       "InstE2MenergyMeterDriver".driverData.pL1Min := 0.0;
       "InstE2MenergyMeterDriver".driverData.pL1Max := 0.0;
       "InstE2MenergyMeterDriver".driverData.pL2Min := 0.0;
       "InstE2MenergyMeterDriver".driverData.pL2Max := 0.0;
       "InstE2MenergyMeterDriver".driverData.pL3Min := 0.0;
       "InstE2MenergyMeterDriver".driverData.pL3Max := 0.0;

       "InstE2MenergyMeterDriver".driverData.qL1Min := 0.0;
       "InstE2MenergyMeterDriver".driverData.qL1Max := 0.0;
       "InstE2MenergyMeterDriver".driverData.qL2Min := 0.0;
       "InstE2MenergyMeterDriver".driverData.qL2Max := 0.0;
       "InstE2MenergyMeterDriver".driverData.qL3Min := 0.0;
       "InstE2MenergyMeterDriver".driverData.qL3Max := 0.0;

   END_IF;

   "Unit1.EmNodes".powerMeter := "InstE2MenergyMeterDriver".driverData;
END_REGION

REGION Network 4: Routing AI_EnergyMeter data to HMI interface
   // Call of Lsicar_EnMeterDataToHmi FB
   RUNG wire#powerrail
      "InstEmDataHmi"(energyMeter01Visu := "InstE2MenergyMeterDriver".driverData, energyMeter02Visu :=, energyMeter03Visu :=, energyMeter04Visu :=, energyMeter05Visu :=, energyMeter06Visu :=, energyMeter07Visu :=, energyMeter08Visu :=)
   END_RUNG
   // the same network as SCL:
   "InstEmDataHmi"(energyMeter01Visu := "InstE2MenergyMeterDriver".driverData);   // "LSicar_EnMeterDataToHmi"
END_REGION
END_FUNCTION

FUNCTION "CallEnEffMonitor" : Void   // FC32, LAD
TITLE = CallEnergyEfficencyMonitor
AUTHOR : SICAR
FAMILY : Energy_EEM
VERSION : 1.0
// The S7 Energy Efficiency-Monitor (or S7 EE-Monitor) allows you to record the energy consumption of your machine in a SIMATIC controller, and to analyze the results on the basis of the energy and media requirements.
// stored: IsIECCheckEnabled true, SetENOAutomatically true
   VAR_TEMP
      tempMeasPointIndex : USInt;   // HMI index
      tempCycleCounterAvgCalc : DInt;   // Calculation to TOD
      tempPlantInProduction : Bool;   // Plant in production
      tempReturnValue : Int;   // Temporärer Wert zur Speicherung der EnPi-Resetzeit
   END_VAR
   // Ret_Val : Ret_Val
   VAR_TEMP   // added for the SCL form of the ladder/FBD networks
      _w1 : Bool;
      _w2 : Bool;
      _w3 : Bool;
      _w4 : Bool;
   END_VAR
BEGIN

REGION Network 1: BLOCK INFO HEADER
   // SIEMENS AG / (c)Copyright 2023
   // ------------------------------------------------------------------------------
   // Title:            CallEnEffMonitor (FC32)
   // Comment/Function: Call of Demo EnergyMeter and Energy Efficient M for EEMM demonstration
   // Library/Family:   Energy
   // Author:           SICAR
   // Tested with:      ---
   // Engineering:      TIA Portal V19
   // Restrictions:     -
   // Requirements:     ---
   // ------------------------------------------------------------------------------
   // Change log table:
   // Version  | Date       | Expert in charge       | Changes applied
   // ---------|------------|------------------------|------------------------------
   // 05.00.00 | 01.09.2023 | SICAR
   //                         First released version
END_REGION

REGION Network 2: DESCRIPTION
   // The Energy Efficiency Monitor “EEM” integrated in SICAR is based on the application example in entry ID: 109753230 V1.0 dated 02/2018 of the Siemens Industry Online Support, see: 
   // 
   // https://support.industry.siemens.com/cs/document/109753230/-s7-energy-efficiency-monitor-for-machines?dti=0&lc=en-WW 
   // 
   // **License**  
   // The software package has to be licensed. The necessary license key has to be entered in the data block for energy data “EEmData”, in the array item “licenseKey”. 
   //  
   // {.pageWidth}
   // ![Image](EemEnPiCalc/en/image1.PNG)
   // 
   // The S7 Energy Efficiency-Monitor (or S7 EE-Monitor) allows you to record the energy consumption of your machine in a SIMATIC controller, and to analyze the results on the basis of the energy and media requirements.  
   // https://support.industry.siemens.com/cs/document/109753230/s7-energieeffizienz-monitor-für-maschinen?dti=0&lc=de-WW 
   // 
   // **PLC Data types**  
   //  LSicar_typeEeMenPiCalc 
   //  LSicar_typeEeMenPiEstate 
   //  LSicar_typeEeMenPiLimit 
   //  typeEnMeterOutputData 
   //  typeMeasDataProfileE3 
   //  
   // **WinCC Faceplates**  
   // 
   // ![Image](EemEnPiCalc/en/image3.PNG)
   // 
   // **WinCC Screen**  
   //  
   // ![Image](EemEnPiCalc/en/image4.PNG)
   //  
   // # Devices & networks 
   // 
   // An additional AI Energy Meter has been added and configured in the SICAR project. The user data has been  
   // configured as module version “EE@Industry measured data profile e3”.  
   // 
   // Select the module version according to your requirements. The data assignment in the FC blocks has to be adjusted according to the selected module version. 
   // 
   // ![Image](EemEnPiCalc/en/image5.PNG)
   //  
   //  
   // 
   //  #### PLC Programm blocks 
   // 
   // ##### CallEnSeem  
   // The block is called in OB “CYCLIC_INTERRUPT_100MS_OB” (100ms cycle). The block contains the following instructions which can be found in “Instructions > Optional packages > Energy Suite extensions”.
   // 
   // **EnS_EEm_Calc:**  
   // The instruction calculates operating state-related energy data of machines and plants for uniform efficiency evaluation, in accordance with the VDMA 34179 measuring directive. 
   // 
   // ---
   // Note
   // :     The instruction calculates the energy efficiency value of the respective state for up to 8 operating states, and the global energy efficiency value. 
   // :     The maximum number of configurable measuring points is 10. Refer to the documentation of the entry ID. 
   // 
   // ---
   // 
   // **EnS_EEm_Report:**  
   // The instruction writes the data for the efficiency report to the data log on the SIMATIC memory card, in accordance with the VDMA 34179 measuring directive. The data log is a CSV file. 
   // 
   // ##### CallEnEffMonitor
   // ---
   // Note
   // :     The assignment of the readings as well as the formation of additional signals can be represented only exemplarily here. It has to be adapted to the actual plant conditions! 
   // 
   // ---
   // 
   // * Networks 1 & 2: The readings of the two AI-Energy-Meters are entered in the DB “EeMonitor”, in an array [0..9] in accordance with the measurement data profile “typeMeasDataProfileE3”. 
   // * Network 3: According to the selection of a measuring point on the HMI, data of the respective measuring point is routed to the HMI data area. The selection is done with a Pull-Down menu and a symbolic I/O field. 
   // * Network 4: Several tags in the EnS…data types are not marked as accessible / visible. In order to display these tags on the HMI all the same, they are routed to DB “EeMonitor” in structure “typeEnMeterWorkHmi”. There the tags are marked as accessible / visible.  
   // * Network 5: A collective signal is generated, according to the exemplary calls for OP area 1. This is only an example! The collective signal shows that the plant is producing parts, by a disjunction (OR) of all outputs. If an output is controlled, the plant is moving and producing parts. This collective signal is used later on to generate the energetic states “eState”. A delay of 3 seconds has been configured so that a short break in controlling the outputs will not change the energetic state. *
   // * Network 6: The signals for the energetic states are generated here. 
   // * Network 7: Simulation On/Off: A part counter is simulated here. Note: the simulation can be switched on and off with a button in the screen. 
   // * Network 8: Simulation On/Off. Energy counters for both AI-Energy-Meters are simulated here. Note: the simulation can be switched on and off with a button in the screen. 
   // * Network 9: Call of blocks “EemDemoSimulation” and “EemDemoResetValEMeter”. 
   // * Network 10: Call of block “EemEnPiCalc” and data routing according to the selection of a measuring point on the HMI. 
   // * Network 11: Error evaluation of block “EemEnPiCalc” to generate ProDiag messages. 
   // * Network 12: Error evaluation of block “EnS_EEm_Report” to generate ProDiag messages.  
   // 
   // ##### EemDemoResetValEMeter  
   // 
   // The block resets certain measurement values by controlling the respective outputs in the I/O area of the AI-Energy-Meter. 
   // 
   // ##### EemDemoSimulation  
   // 
   // This block simulates higher or lower energy values, according to the energetic states “eState”. 
   // 
   // ##### EemEnPiCalc
   // This block calculates the ENPI (Energy value Pro Item). It substitutes the script “EEm_EnPI_Efficiency” of the entry ID. 
   // 
   // ---
   // Note
   // :     All block parameters are provided with “pre-defined actual parameters”.
   // 
   // ---
   // 
   // **Operation mode Automatic / Manual**  
   // 
   // The blocks are independent of operation modes. Therefor they are not assigned to any operation mode area. 
   // 
   // **PLC Alarm text list**  
   // 
   // The following PLC alarm text lists have been created: 
   // 
   // * **EEMonitor_Calc_Warn_PD** ProDiag alarm text list for alarms by instruction “EnS_EEm_Calc”.   
   // * **EEMonitor_Report_Warn_PD** ProDiag alarm text list for alarms by instruction “EnS_EEm_Report”.   
   // Both PLC alarm text lists have been entered in the PLC alarm text list “GLOBAL_GENERAL_AlarmTextList”. 
   // 
   // ---
   // Note
   // :     The alarm texts are provided in two languages (German, English). Please consider the multilingual nature of the entries. 
   // 
   // ---
   // 
   // #### PLC Data types 
   // 
   // PLC data types used for PLC program block or HMI faceplate:  
   // ![Image](_Icon/reference.PNG)  See ..\Library Types\LSicar_typeEeMenPiCalc.pdf  
   // 
   // #### WinCC Objects 
   // 
   // **WinCC HMI-tags**  
   // 
   // The HMI tags are stored in the tag table “AI_EnergyMeter_EEM” in the SICAR project.  
   // 
   // **WinCC Text and graphics lists**  
   // 
   // The text list “EE-MONITOR_MEASUREPOINT” contains the texts necessary for the pull-down menu / symbolic I/O field in the screen. Please take into account the multilingual nature of the entries.  
   // 
   // **WinCC Faceplates**  
   // 
   // The faceplates are stored in the project library, in folder “types”. They have been created using several WinCC objects; they are animated depending on the state. 
   // 
   // * EEM_EnPI_EnergyPerItem:	display of ENPI (ENergy Per Item) 
   // * EEM_ViewBar_Diff-AVG-REF:	bar display to compare reference value and average value 
   // * EEM_ViewBar_EState-Total:	bar display of energy status (not used at this time) 
   // * EEM_ViewBarCurve_EState:	Total: bar display and curve display of the energy values  
   // 
   // **WinCC-screen** 
   // 
   // 1. HMI Screens:	EE-MONITOR_ENERGY: display of the energy values 
   // 2. HMI Popup-screens 
   // 	* EEM_LEGEND_Popup: 		Legend 
   // 	* EEM_INFO-MACHINE_Popup: 	Machine information 
   // 	* EEM_STARTMEASURE_Popup: 	Popup to start the normal measurement or the reference measurement  
   // 	* EEM_UIPE_Popup: 		display of voltage, current, power, and energy 
   // 	* MORE_EEM_Popup: 		Popup with additional buttons 
   // 	* MORE_AddOn_Popup: 		supplemented  with button “EE-Monitor” 
   // 
   //  
   // 
   // {.pageWidth}
   // ![Image](EemEnPiCalc/en/image6.PNG)
   //  
   //  
   // 
   // #### Additional information
   // 
   // #### Update info
   // 
   // #### Further documentations
END_REGION

REGION Network 3: select measurement values
   // can be from EnergyMeter driver or directly from any hardware (in this example EnergyMeter module and PAC)
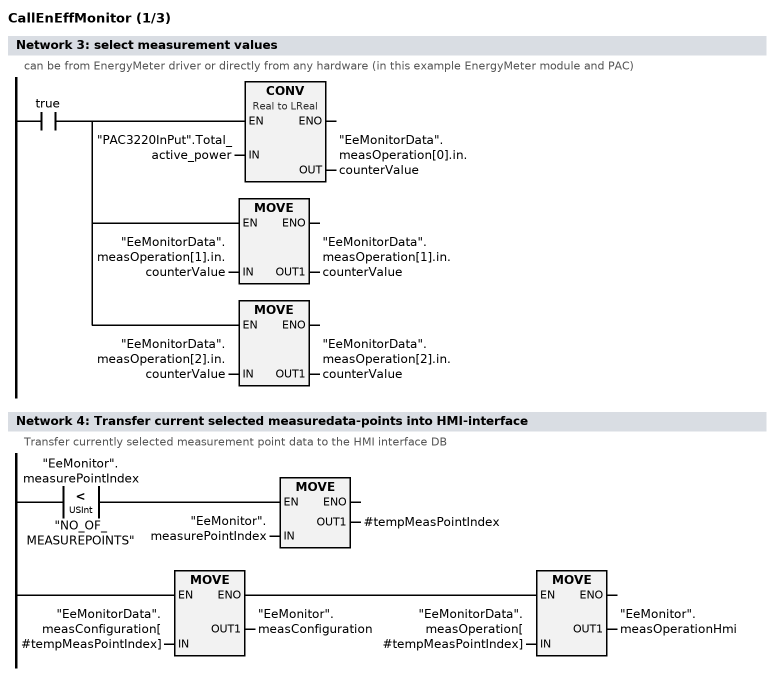
   RUNG wire#powerrail
      Contact( true )
      wire#w1
      { S7_Templates := "[SrcType := Real, DestType := LReal]" } Convert(in := "PAC3220InPut".Total_active_power, out => "EeMonitorData".measOperation[0].in.counterValue)
   END_RUNG
   RUNG wire#w1
      Move(in := "EeMonitorData".measOperation[1].in.counterValue, out1 => "EeMonitorData".measOperation[1].in.counterValue)
   END_RUNG
   RUNG wire#w1
      Move(in := "EeMonitorData".measOperation[2].in.counterValue, out1 => "EeMonitorData".measOperation[2].in.counterValue)
   END_RUNG
   // the same network as SCL:
   IF true THEN
       "EeMonitorData".measOperation[0].in.counterValue := REAL_TO_LREAL("PAC3220InPut".Total_active_power);
       "EeMonitorData".measOperation[1].in.counterValue := "EeMonitorData".measOperation[1].in.counterValue;
       "EeMonitorData".measOperation[2].in.counterValue := "EeMonitorData".measOperation[2].in.counterValue;
   END_IF;
END_REGION

REGION Network 4: Transfer current selected measuredata-points into HMI-interface
   // Transfer currently selected measurement point data to the HMI interface DB
   RUNG wire#powerrail
      { S7_Templates := "SrcType := USInt" } LT_Contact(in1 := "EeMonitor".measurePointIndex, in2 := "NO_OF_MEASUREPOINTS")
      Move(in := "EeMonitor".measurePointIndex, out1 => #tempMeasPointIndex)
   END_RUNG
   RUNG wire#powerrail
      Move(in := "EeMonitorData".measConfiguration[#tempMeasPointIndex], out1 => "EeMonitor".measConfiguration)
      Move(in := "EeMonitorData".measOperation[#tempMeasPointIndex], out1 => "EeMonitor".measOperationHmi)
   END_RUNG
   // the same network as SCL:
   IF "EeMonitor".measurePointIndex < "NO_OF_MEASUREPOINTS" THEN
       #tempMeasPointIndex := "EeMonitor".measurePointIndex;
   END_IF;
   "EeMonitor".measConfiguration := "EeMonitorData".measConfiguration[#tempMeasPointIndex];
   "EeMonitor".measOperationHmi := "EeMonitorData".measOperation[#tempMeasPointIndex];
END_REGION

REGION Network 5: WORKaround: Transfer data from EeMonitroData to EeMonitor.work
   // Convertion of Time to DTL and adding time zone with date and time taken from EnS_EEm_Calc for representing the actual date and time in the current country.
   // Data is copied from EeMonitorData to EeMonitor.work
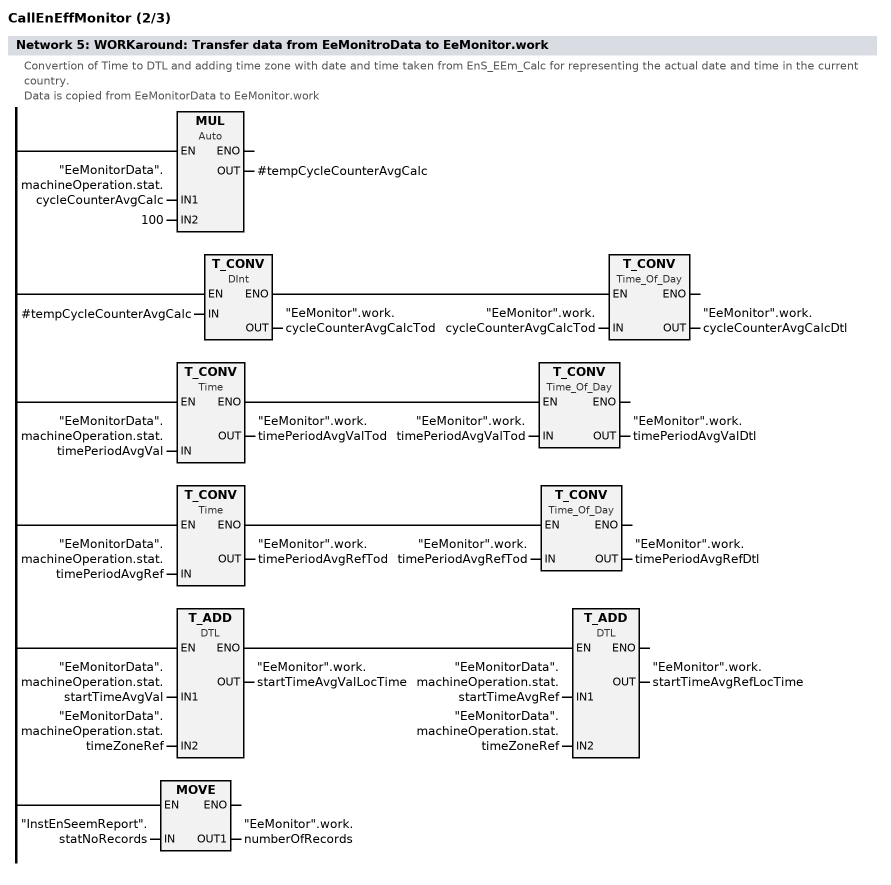
   RUNG wire#powerrail
      Mul(in1 := "EeMonitorData".machineOperation.stat.cycleCounterAvgCalc, in2 := 100, out => #tempCycleCounterAvgCalc)
   END_RUNG
   RUNG wire#powerrail
      { S7_Templates := "[src_type := DInt, dest_type := Time_Of_Day]" } T_CONV(IN := #tempCycleCounterAvgCalc, OUT => "EeMonitor".work.cycleCounterAvgCalcTod)
      { S7_Templates := "[src_type := Time_Of_Day, dest_type := DTL]" } T_CONV(IN := "EeMonitor".work.cycleCounterAvgCalcTod, OUT => "EeMonitor".work.cycleCounterAvgCalcDtl)
   END_RUNG
   RUNG wire#powerrail
      { S7_Templates := "[src_type := Time, dest_type := Time_Of_Day]" } T_CONV(IN := "EeMonitorData".machineOperation.stat.timePeriodAvgVal, OUT => "EeMonitor".work.timePeriodAvgValTod)
      { S7_Templates := "[src_type := Time_Of_Day, dest_type := DTL]" } T_CONV(IN := "EeMonitor".work.timePeriodAvgValTod, OUT => "EeMonitor".work.timePeriodAvgValDtl)
   END_RUNG
   RUNG wire#powerrail
      { S7_Templates := "[src_type := Time, dest_type := Time_Of_Day]" } T_CONV(IN := "EeMonitorData".machineOperation.stat.timePeriodAvgRef, OUT => "EeMonitor".work.timePeriodAvgRefTod)
      { S7_Templates := "[src_type := Time_Of_Day, dest_type := DTL]" } T_CONV(IN := "EeMonitor".work.timePeriodAvgRefTod, OUT => "EeMonitor".work.timePeriodAvgRefDtl)
   END_RUNG
   RUNG wire#powerrail
      { S7_Templates := "[date_type := DTL, time_type := Time]" } T_ADD(IN1 := "EeMonitorData".machineOperation.stat.startTimeAvgVal, IN2 := "EeMonitorData".machineOperation.stat.timeZoneRef, OUT => "EeMonitor".work.startTimeAvgValLocTime)
      { S7_Templates := "[date_type := DTL, time_type := Time]" } T_ADD(IN1 := "EeMonitorData".machineOperation.stat.startTimeAvgRef, IN2 := "EeMonitorData".machineOperation.stat.timeZoneRef, OUT => "EeMonitor".work.startTimeAvgRefLocTime)
   END_RUNG
   RUNG wire#powerrail
      Move(in := "InstEnSeemReport".statNoRecords, out1 => "EeMonitor".work.numberOfRecords)
   END_RUNG
   // the same network as SCL:
   #tempCycleCounterAvgCalc := "EeMonitorData".machineOperation.stat.cycleCounterAvgCalc * 100;
   T_CONV(IN := #tempCycleCounterAvgCalc, OUT => "EeMonitor".work.cycleCounterAvgCalcTod, ENO => #_w1);
   IF #_w1 THEN
       T_CONV(IN := "EeMonitor".work.cycleCounterAvgCalcTod, OUT => "EeMonitor".work.cycleCounterAvgCalcDtl);
   END_IF;
   T_CONV(IN := "EeMonitorData".machineOperation.stat.timePeriodAvgVal,
          OUT => "EeMonitor".work.timePeriodAvgValTod,
          ENO => #_w2);
   IF #_w2 THEN
       T_CONV(IN := "EeMonitor".work.timePeriodAvgValTod, OUT => "EeMonitor".work.timePeriodAvgValDtl);
   END_IF;
   T_CONV(IN := "EeMonitorData".machineOperation.stat.timePeriodAvgRef,
          OUT => "EeMonitor".work.timePeriodAvgRefTod,
          ENO => #_w3);
   IF #_w3 THEN
       T_CONV(IN := "EeMonitor".work.timePeriodAvgRefTod, OUT => "EeMonitor".work.timePeriodAvgRefDtl);
   END_IF;
   T_ADD(IN1 := "EeMonitorData".machineOperation.stat.startTimeAvgVal,
         IN2 := "EeMonitorData".machineOperation.stat.timeZoneRef,
         OUT => "EeMonitor".work.startTimeAvgValLocTime,
         ENO => #_w4);
   IF #_w4 THEN
       T_ADD(IN1 := "EeMonitorData".machineOperation.stat.startTimeAvgRef,
             IN2 := "EeMonitorData".machineOperation.stat.timeZoneRef,
             OUT => "EeMonitor".work.startTimeAvgRefLocTime);
   END_IF;
   "EeMonitor".work.numberOfRecords := "InstEnSeemReport".statNoRecords;
END_REGION

REGION Network 6: Operation modes to "eState"
   // Sets Estate number accoriding to the selected state
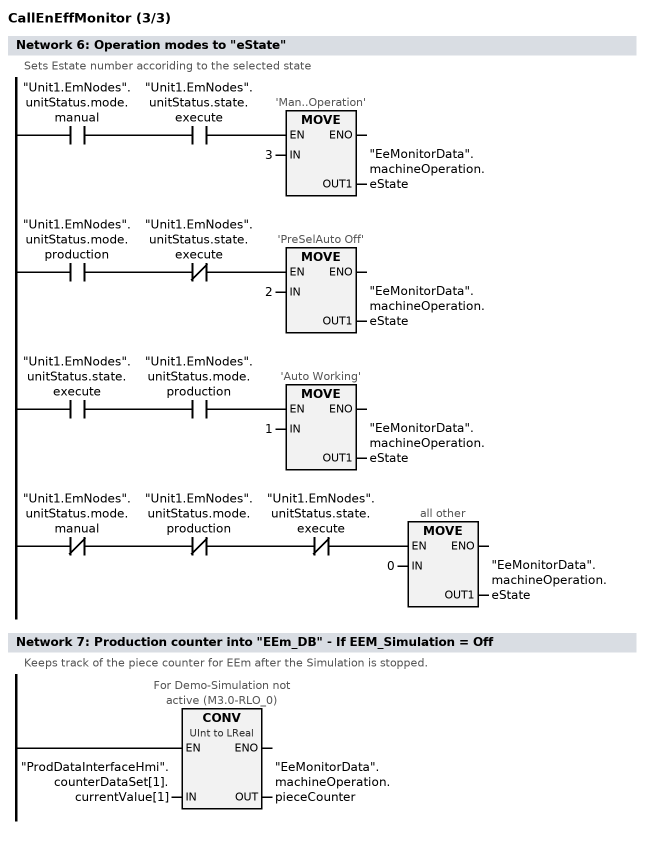
   RUNG wire#powerrail
      Contact( "Unit1.EmNodes".unitStatus.mode.manual )
      Contact( "Unit1.EmNodes".unitStatus.state.execute )
      Move(in := 3, out1 => "EeMonitorData".machineOperation.eState)   // 'Man..Operation'
   END_RUNG
   RUNG wire#powerrail
      Contact( "Unit1.EmNodes".unitStatus.mode.production )
      I_Contact( "Unit1.EmNodes".unitStatus.state.execute )
      Move(in := 2, out1 => "EeMonitorData".machineOperation.eState)   // 'PreSelAuto Off'
   END_RUNG
   RUNG wire#powerrail
      Contact( "Unit1.EmNodes".unitStatus.state.execute )
      Contact( "Unit1.EmNodes".unitStatus.mode.production )
      Move(in := 1, out1 => "EeMonitorData".machineOperation.eState)   // 'Auto Working'
   END_RUNG
   RUNG wire#powerrail
      I_Contact( "Unit1.EmNodes".unitStatus.mode.manual )
      I_Contact( "Unit1.EmNodes".unitStatus.mode.production )
      I_Contact( "Unit1.EmNodes".unitStatus.state.execute )
      Move(in := 0, out1 => "EeMonitorData".machineOperation.eState)   // all other
   END_RUNG
   // the same network as SCL:
   IF "Unit1.EmNodes".unitStatus.mode.manual AND "Unit1.EmNodes".unitStatus.state.execute THEN
       "EeMonitorData".machineOperation.eState := 3;   // 'Man..Operation'
   END_IF;
   IF "Unit1.EmNodes".unitStatus.mode.production AND NOT "Unit1.EmNodes".unitStatus.state.execute THEN
       "EeMonitorData".machineOperation.eState := 2;   // 'PreSelAuto Off'
   END_IF;
   IF "Unit1.EmNodes".unitStatus.state.execute AND "Unit1.EmNodes".unitStatus.mode.production THEN
       "EeMonitorData".machineOperation.eState := 1;   // 'Auto Working'
   END_IF;
   IF NOT "Unit1.EmNodes".unitStatus.mode.manual AND NOT "Unit1.EmNodes".unitStatus.mode.production AND NOT "Unit1.EmNodes".unitStatus.state.execute THEN
       "EeMonitorData".machineOperation.eState := 0;   // all other
   END_IF;
END_REGION

REGION Network 7: Production counter into "EEm_DB" - If EEM_Simulation = Off
   // Keeps track of the piece counter for EEm after the Simulation is stopped.
   RUNG wire#powerrail
      { S7_Templates := "[SrcType := UInt, DestType := LReal]" } Convert(in := "ProdDataInterfaceHmi".counterDataSet[1].currentValue[1], out => "EeMonitorData".machineOperation.pieceCounter)   // For Demo-Simulation not active (M3.0-RLO_0)
   END_RUNG
   // the same network as SCL:
   "EeMonitorData".machineOperation.pieceCounter := UINT_TO_LREAL("ProdDataInterfaceHmi".counterDataSet[1].currentValue[1]);   // For Demo-Simulation not active (M3.0-RLO_0)
END_REGION

REGION Network 8 (SCL): Reset EnPI values
   // Reads the current time and store it to provide the user the information about the last EnPi reset
   // Check for the trigger to reset/recalculate the EnPI values
   IF ("EeMonitorData".internalData.enpiResetTrigger = TRUE) THEN

       // Read the current time and store it to provide the user the information
       // about the last reset
       #tempReturnValue := RD_LOC_T("EeMonitorData".internalData.enpiResetTime);

       // Reset the trigger
       "EeMonitorData".internalData.enpiResetTrigger := FALSE;
   ELSE
       ; // No trigger
   END_IF;
END_REGION
END_FUNCTION

FUNCTION "CallSettings" : Void   // FC8, LAD
// Call of settings blocks
// stored: IsIECCheckEnabled true, SetENOAutomatically false
BEGIN

REGION Network 1: BLOCK INFO HEADER
   // SIEMENS AG / (c)Copyright 2023
   // ------------------------------------------------------------------------------
   // Title:            CallSettings
   // Comment/Function: Call of SICAR Settings blocks
   // Library/Family:   -
   // Author:           -
   // Tested with:      ---
   // Engineering:      TIA Portal V19
   // Restrictions:     -
   // Requirements:     ---
   // ------------------------------------------------------------------------------
   // Change log table:
   // Version | Date | Expert in charge | Changes applied
   // -------|---------|-------------|--------------------------------------------
   // 01.00.00 | 01.01.1999 | Person x | First released version
   // 01.00.01 | 02.01.1999 | Person y | Block was Updated
END_REGION

REGION Network 2: Set set PLC date and time
   // Change local date and time of the PLC
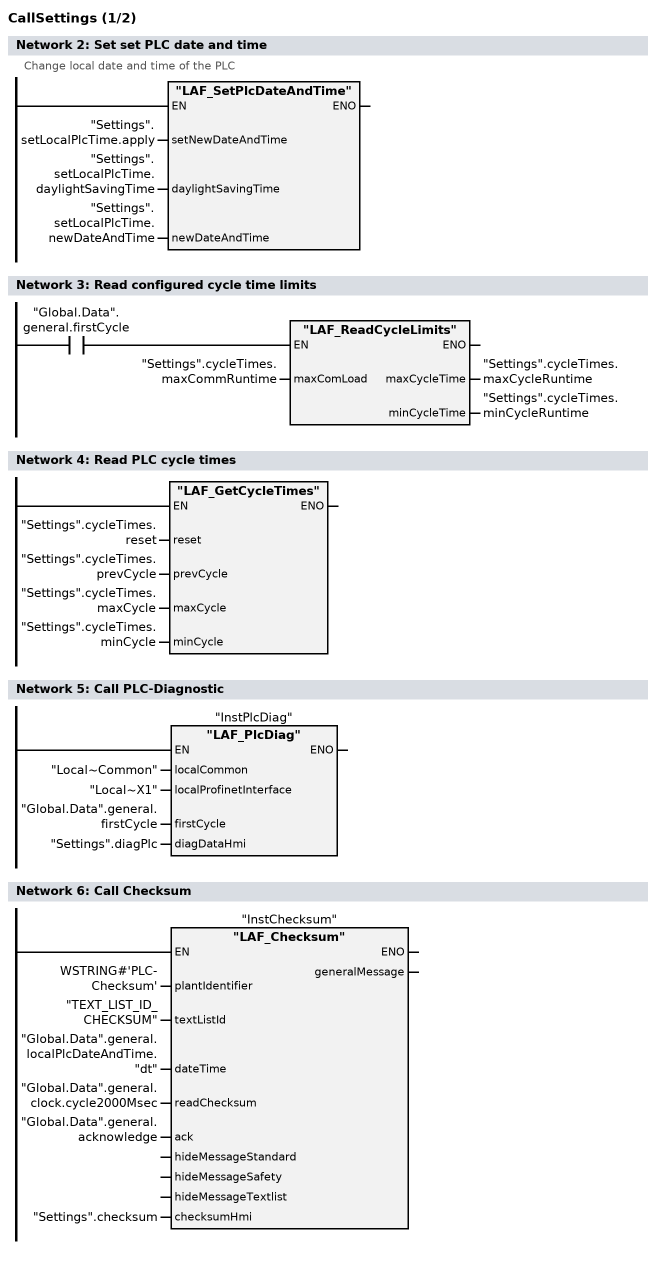
   RUNG wire#powerrail
      "LAF_SetPlcDateAndTime"(setNewDateAndTime := "Settings".setLocalPlcTime.apply, daylightSavingTime := "Settings".setLocalPlcTime.daylightSavingTime, newDateAndTime := "Settings".setLocalPlcTime.newDateAndTime)
   END_RUNG
   // the same network as SCL:
   "LAF_SetPlcDateAndTime"(setNewDateAndTime := "Settings".setLocalPlcTime.apply,
                           daylightSavingTime := "Settings".setLocalPlcTime.daylightSavingTime,
                           newDateAndTime := "Settings".setLocalPlcTime.newDateAndTime);
END_REGION

REGION Network 3: Read configured cycle time limits
   RUNG wire#powerrail
      Contact( "Global.Data".general.firstCycle )
      "LAF_ReadCycleLimits"(maxComLoad := "Settings".cycleTimes.maxCommRuntime, maxCycleTime => "Settings".cycleTimes.maxCycleRuntime, minCycleTime => "Settings".cycleTimes.minCycleRuntime)
   END_RUNG
   // the same network as SCL:
   IF "Global.Data".general.firstCycle THEN
       "LAF_ReadCycleLimits"(maxComLoad := "Settings".cycleTimes.maxCommRuntime,
                             maxCycleTime => "Settings".cycleTimes.maxCycleRuntime,
                             minCycleTime => "Settings".cycleTimes.minCycleRuntime);
   END_IF;
END_REGION

REGION Network 4: Read PLC cycle times
   RUNG wire#powerrail
      "LAF_GetCycleTimes"(reset := "Settings".cycleTimes.reset, prevCycle := "Settings".cycleTimes.prevCycle, maxCycle := "Settings".cycleTimes.maxCycle, minCycle := "Settings".cycleTimes.minCycle)
   END_RUNG
   // the same network as SCL:
   "LAF_GetCycleTimes"(reset := "Settings".cycleTimes.reset,
                       prevCycle := "Settings".cycleTimes.prevCycle,
                       maxCycle := "Settings".cycleTimes.maxCycle,
                       minCycle := "Settings".cycleTimes.minCycle);
END_REGION

REGION Network 5: Call PLC-Diagnostic
   RUNG wire#powerrail
      "InstPlcDiag"(localCommon := "Local~Common", localProfinetInterface := "Local~X1", firstCycle := "Global.Data".general.firstCycle, diagDataHmi := "Settings".diagPlc)
   END_RUNG
   // the same network as SCL:
   "InstPlcDiag"(localCommon := "Local~Common",   // "LAF_PlcDiag"
                 localProfinetInterface := "Local~X1",
                 firstCycle := "Global.Data".general.firstCycle,
                 diagDataHmi := "Settings".diagPlc);
END_REGION

REGION Network 6: Call Checksum
   RUNG wire#powerrail
      "InstChecksum"(plantIdentifier := WSTRING#'PLC-Checksum', textListId := "TEXT_LIST_ID_CHECKSUM", dateTime := "Global.Data".general.localPlcDateAndTime."dt", readChecksum := "Global.Data".general.clock.cycle2000Msec, ack := "Global.Data".general.acknowledge, hideMessageStandard :=, hideMessageSafety :=, hideMessageTextlist :=, checksumHmi := "Settings".checksum, generalMessage =>)
   END_RUNG
   // the same network as SCL:
   "InstChecksum"(plantIdentifier := WSTRING#'PLC-Checksum',   // "LAF_Checksum"
                  textListId := "TEXT_LIST_ID_CHECKSUM",
                  dateTime := "Global.Data".general.localPlcDateAndTime."dt",
                  readChecksum := "Global.Data".general.clock.cycle2000Msec,
                  ack := "Global.Data".general.acknowledge,
                  checksumHmi := "Settings".checksum);
END_REGION

REGION Network 7: Call SMC-Diagnostic (SIMATIC Memory Card - Diagnostic)
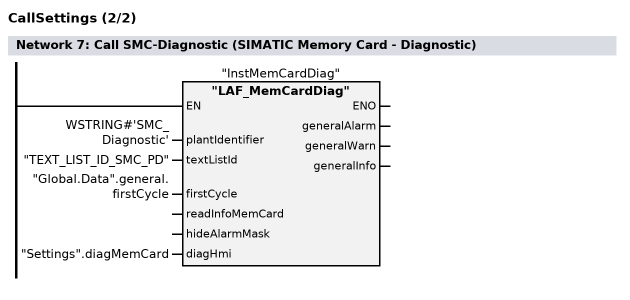
   RUNG wire#powerrail
      "InstMemCardDiag"(plantIdentifier := WSTRING#'SMC_Diagnostic', textListId := "TEXT_LIST_ID_SMC_PD", firstCycle := "Global.Data".general.firstCycle, readInfoMemCard :=, hideAlarmMask :=, diagHmi := "Settings".diagMemCard, generalAlarm =>, generalWarn =>, generalInfo =>)
   END_RUNG
   // the same network as SCL:
   "InstMemCardDiag"(plantIdentifier := WSTRING#'SMC_Diagnostic',   // "LAF_MemCardDiag"
                     textListId := "TEXT_LIST_ID_SMC_PD",
                     firstCycle := "Global.Data".general.firstCycle,
                     diagHmi := "Settings".diagMemCard);
END_REGION
END_FUNCTION

ORGANIZATION_BLOCK "DiagnosticErrorInterrupt"   // OB82, LAD, DiagnosticErrorInterrupt
// stored: SetENOAutomatically false
   VAR_INPUT
      IO_State : Word;   // IO state of the HW object
      LADDR : HW_ANY;   // Hardware identifier
      Channel : UInt;   // Channel number
      MultiError : Bool;   // =true if more than one error is present
   END_VAR
BEGIN
END_ORGANIZATION_BLOCK

ORGANIZATION_BLOCK "HardwareInterrupt"   // OB40, LAD, HardwareInterrupt
// stored: SetENOAutomatically false
   VAR_INPUT
      LADDR : HW_IO;   // Hardware identifier
      USI : Word;   // User structure identifier
      IChannel : USInt;   // Interrupt channel number
      EventType : Byte;   // EventType
      PointAddr : DWord;
   END_VAR
BEGIN
END_ORGANIZATION_BLOCK

ORGANIZATION_BLOCK "IO_AccessError"   // OB122, LAD, IOAccessError
// stored: SetENOAutomatically false
   VAR_INPUT
      BlockNr : UInt;   // Number of causing block
      Reaction : USInt;   // 0:ignore, 1:substitute, 2:skip
      Fault_ID : Byte;   // 16#42:reading, 16#43:writing
      BlockType : USInt;   // 16#01:OB, 16#02:FC, 16#03:FB, 16#04:SFC, 16#05:SFB, 16#06:DB: Type of block causing the error
      Area : USInt;   // 16#81:I, 16#82:Q: IO area where the IOaccess error occured
      DBNr : DB_ANY;   // Reserved for system
      Csg_OBNr : OB_ANY;   // Number of OB causing the error
      Csg_Prio : USInt;   // Priority of OB causing the error
      Width : USInt;   // 0:bit, 1:byte, 2:word, 3:dword, 4:lword
   END_VAR
BEGIN
END_ORGANIZATION_BLOCK

ORGANIZATION_BLOCK "Interrupt1s"   // OB31, LAD, CyclicInterrupt
TITLE = Cyclic interrupt 100ms
AUTHOR : SICAR
FAMILY : OB
VERSION : 1.0
// organisation block
// stored: IsIECCheckEnabled true, SetENOAutomatically true
   VAR_INPUT
      Initial_Call : Bool;   // Initial call of this OB
      Event_Count : Int;   // Events discarded
   END_VAR
BEGIN

REGION Network 1: ChangeLog
   // Change log table:
   // Version | Date | Expert in charge | Changes applied
   // -------|---------|-------------|--------------------------------------------
   // 01.00.00 | 01.01.1999 | Person x | First released version
   // 01.00.01 | 02.01.1999 | Person y | Block was Updated
END_REGION

REGION Network 2: Call & measure-data into "EEmData_DB"
   // Call the energy efficiency monitor functions
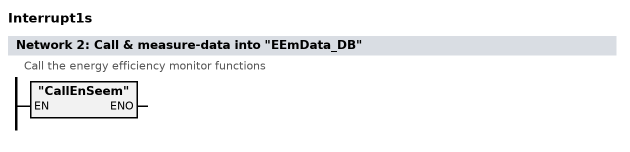
   RUNG wire#powerrail
      "CallEnSeem"()
   END_RUNG
   // the same network as SCL:
   "CallEnSeem"();
END_REGION
END_ORGANIZATION_BLOCK

FUNCTION "CallEnSeem" : Void   // FC34, LAD
TITLE = CallEnSeem
AUTHOR : SICAR
FAMILY : Energy_EEM
VERSION : 1.0
// The S7 Energy Efficiency-Monitor (or S7 EE-Monitor) allows you to record the energy consumption of your machine in a SIMATIC controller, and to analyze the results on the basis of the energy and media requirements.
// stored: IsIECCheckEnabled true, SetENOAutomatically true
   // Ret_Val : Ret_Val
BEGIN

REGION Network 1: BLOCK INFO HEADER
   // SIEMENS AG / (c)Copyright 2023
   // ------------------------------------------------------------------------------
   // Title:            CallEnSeem (FC34)
   // Comment/Function: The S7 Energy Efficiency-Monitor (or S7 EE-Monitor) allows you to record the energy consumption of your machine in a SIMATIC controller, and to analyze the results on the basis of the energy and media requirements.
   // Library/Family:   Energy_EEM
   // Author:           SICAR
   // Tested with:      ---
   // Engineering:      TIA Portal V19
   // Restrictions:     -
   // Requirements:     ---
   // ------------------------------------------------------------------------------
   // Change log table:
   // Version | Date | Expert in charge | Changes applied
   // -------|---------|-------------|--------------------------------------------
   // 01.00.00 | 01.01.1999 | Person x | First released version
   // 01.00.01 | 02.01.1999 | Person y | Block was Updated
END_REGION

REGION Network 2: DESCRIPTION
   // The Energy Efficiency Monitor “EEM” integrated in SICAR is based on the application example in entry ID: 109753230 V1.0 dated 02/2018 of the Siemens Industry Online Support, see: 
   // 
   // https://support.industry.siemens.com/cs/document/109753230/-s7-energy-efficiency-monitor-for-machines?dti=0&lc=en-WW 
   // 
   // **License**  
   // The software package has to be licensed. The necessary license key has to be entered in the data block for energy data “EEmData”, in the array item “licenseKey”. 
   //  
   // {.pageWidth}
   // ![Image](EemEnPiCalc/en/image1.PNG)
   // 
   // The S7 Energy Efficiency-Monitor (or S7 EE-Monitor) allows you to record the energy consumption of your machine in a SIMATIC controller, and to analyze the results on the basis of the energy and media requirements.  
   // https://support.industry.siemens.com/cs/document/109753230/s7-energieeffizienz-monitor-für-maschinen?dti=0&lc=de-WW 
   // 
   // **PLC Data types**  
   //  LSicar_typeEeMenPiCalc 
   //  LSicar_typeEeMenPiEstate 
   //  LSicar_typeEeMenPiLimit 
   //  typeEnMeterOutputData 
   //  typeMeasDataProfileE3 
   //  
   // **WinCC Faceplates**  
   // 
   // ![Image](EemEnPiCalc/en/image3.PNG)
   // 
   // **WinCC Screen**  
   //  
   // ![Image](EemEnPiCalc/en/image4.PNG)
   //  
   // # Devices & networks 
   // 
   // An additional AI Energy Meter has been added and configured in the SICAR project. The user data has been  
   // configured as module version “EE@Industry measured data profile e3”.  
   // 
   // Select the module version according to your requirements. The data assignment in the FC blocks has to be adjusted according to the selected module version. 
   // 
   // ![Image](EemEnPiCalc/en/image5.PNG)
   //  
   //  
   // 
   // #### PLC Programm blocks 
   // 
   // ##### CallEnSeem  
   // The block is called in OB “CYCLIC_INTERRUPT_100MS_OB” (100ms cycle). The block contains the following instructions which can be found in “Instructions > Optional packages > Energy Suite extensions”.
   // 
   // **EnS_EEm_Calc:**  
   // The instruction calculates operating state-related energy data of machines and plants for uniform efficiency evaluation, in accordance with the VDMA 34179 measuring directive. 
   // 
   // ---
   // Note
   // :     The instruction calculates the energy efficiency value of the respective state for up to 8 operating states, and the global energy efficiency value. 
   // :     The maximum number of configurable measuring points is 10. Refer to the documentation of the entry ID. 
   // 
   // ---
   // 
   // **EnS_EEm_Report:**  
   // The instruction writes the data for the efficiency report to the data log on the SIMATIC memory card, in accordance with the VDMA 34179 measuring directive. The data log is a CSV file. 
   // 
   // #### CallEnEffMonitor
   // ---
   // Note
   // :     The assignment of the readings as well as the formation of additional signals can be represented only exemplarily here. It has to be adapted to the actual plant conditions! 
   // 
   // ---
   // 
   // * Networks 1 & 2: The readings of the two AI-Energy-Meters are entered in the DB “EeMonitor”, in an array [0..9] in accordance with the measurement data profile “typeMeasDataProfileE3”. 
   // * Network 3: According to the selection of a measuring point on the HMI, data of the respective measuring point is routed to the HMI data area. The selection is done with a Pull-Down menu and a symbolic I/O field. 
   // * Network 4: Several tags in the EnS…data types are not marked as accessible / visible. In order to display these tags on the HMI all the same, they are routed to DB “EeMonitor” in structure “typeEnMeterWorkHmi”. There the tags are marked as accessible / visible.  
   // * Network 5: A collective signal is generated, according to the exemplary calls for OP area 1. This is only an example! The collective signal shows that the plant is producing parts, by a disjunction (OR) of all outputs. If an output is controlled, the plant is moving and producing parts. This collective signal is used later on to generate the energetic states “eState”. A delay of 3 seconds has been configured so that a short break in controlling the outputs will not change the energetic state. *
   // * Network 6: The signals for the energetic states are generated here. 
   // * Network 7: Simulation On/Off: A part counter is simulated here. Note: the simulation can be switched on and off with a button in the screen. 
   // * Network 8: Simulation On/Off. Energy counters for both AI-Energy-Meters are simulated here. Note: the simulation can be switched on and off with a button in the screen. 
   // * Network 9: Call of blocks “EemDemoSimulation” and “EemDemoResetValEMeter”. 
   // * Network 10: Call of block “EemEnPiCalc” and data routing according to the selection of a measuring point on the HMI. 
   // * Network 11: Error evaluation of block “EemEnPiCalc” to generate ProDiag messages. 
   // * Network 12: Error evaluation of block “EnS_EEm_Report” to generate ProDiag messages.  
   // 
   // #### EemDemoResetValEMeter  
   // 
   // The block resets certain measurement values by controlling the respective outputs in the I/O area of the AI-Energy-Meter. 
   // 
   // #### EemDemoSimulation  
   // 
   // This block simulates higher or lower energy values, according to the energetic states “eState”. 
   // 
   // #### EemEnPiCalc
   // This block calculates the ENPI (Energy value Pro Item). It substitutes the script “EEm_EnPI_Efficiency” of the entry ID. 
   // 
   // ---
   // Note
   // :     All block parameters are provided with “pre-defined actual parameters”.
   // 
   // ---
   // 
   // **Operation mode Automatic / Manual**  
   // 
   // The blocks are independent of operation modes. Therefor they are not assigned to any operation mode area. 
   // 
   // **PLC Alarm text list**  
   // 
   // The following PLC alarm text lists have been created: 
   // 
   // * **EEMonitor_Calc_Warn_PD** ProDiag alarm text list for alarms by instruction “EnS_EEm_Calc”.   
   // * **EEMonitor_Report_Warn_PD** ProDiag alarm text list for alarms by instruction “EnS_EEm_Report”.   
   // Both PLC alarm text lists have been entered in the PLC alarm text list “GLOBAL_GENERAL_AlarmTextList”. 
   // 
   // ---
   // Note
   // :     The alarm texts are provided in two languages (German, English). Please consider the multilingual nature of the entries. 
   // 
   // ---
   // 
   // #### PLC Data types 
   // 
   // PLC data types used for PLC program block or HMI faceplate:  
   // ![Image](_Icon/reference.PNG)  See ..\Library Types\LSicar_typeEeMenPiCalc.pdf  
   // 
   // #### WinCC Objects 
   // 
   // **WinCC HMI-tags**  
   // 
   // The HMI tags are stored in the tag table “AI_EnergyMeter_EEM” in the SICAR project.  
   // 
   // **WinCC Text and graphics lists**  
   // 
   // The text list “EE-MONITOR_MEASUREPOINT” contains the texts necessary for the pull-down menu / symbolic I/O field in the screen. Please take into account the multilingual nature of the entries.  
   // 
   // **WinCC Faceplates**  
   // 
   // The faceplates are stored in the project library, in folder “types”. They have been created using several WinCC objects; they are animated depending on the state. 
   // 
   // * EEM_EnPI_EnergyPerItem:	display of ENPI (ENergy Per Item) 
   // * EEM_ViewBar_Diff-AVG-REF:	bar display to compare reference value and average value 
   // * EEM_ViewBar_EState-Total:	bar display of energy status (not used at this time) 
   // * EEM_ViewBarCurve_EState:	Total: bar display and curve display of the energy values  
   // 
   // **WinCC-screen** 
   // 
   // 1. HMI Screens:	EE-MONITOR_ENERGY: display of the energy values 
   // 2. HMI Popup-screens 
   // 	* EEM_LEGEND_Popup: 		Legend 
   // 	* EEM_INFO-MACHINE_Popup: 	Machine information 
   // 	* EEM_STARTMEASURE_Popup: 	Popup to start the normal measurement or the reference measurement  
   // 	* EEM_UIPE_Popup: 		display of voltage, current, power, and energy 
   // 	* MORE_EEM_Popup: 		Popup with additional buttons 
   // 	* MORE_AddOn_Popup: 		supplemented  with button “EE-Monitor” 
   // 
   //  
   // 
   // {.pageWidth}
   // ![Image](EemEnPiCalc/en/image6.PNG)
   //  
   //  
   // 
   // #### Additional information
   // 
   // #### Update info
   // 
   // #### Further documentations
END_REGION

REGION Network 3: EE-Monitor: "Recalc"
   // Toggle for autom. updating the values in the screen every 2nd cycle (every 200ms)
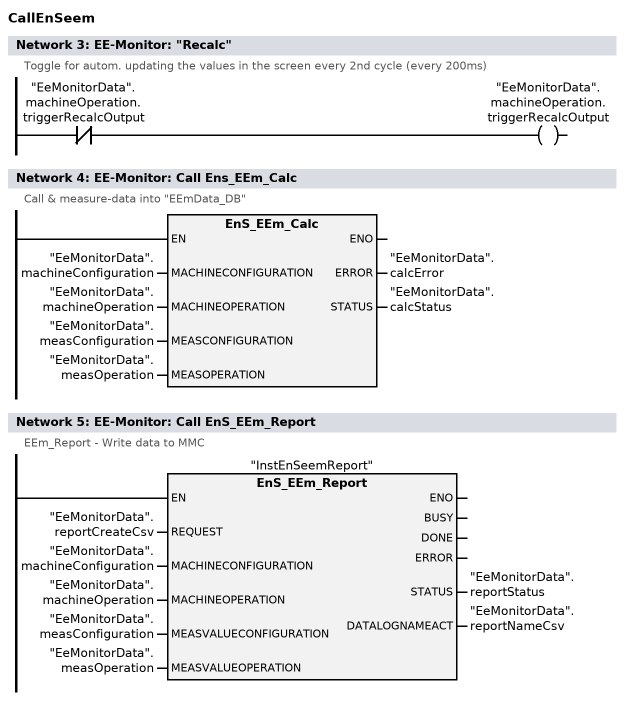
   RUNG wire#powerrail
      I_Contact( "EeMonitorData".machineOperation.triggerRecalcOutput )
      Coil( "EeMonitorData".machineOperation.triggerRecalcOutput )
   END_RUNG
   // the same network as SCL:
   "EeMonitorData".machineOperation.triggerRecalcOutput := NOT "EeMonitorData".machineOperation.triggerRecalcOutput;
END_REGION

REGION Network 4: EE-Monitor: Call Ens_EEm_Calc
   // Call & measure-data into "EEmData_DB"
   RUNG wire#powerrail
      EnS_EEm_Calc(machineConfiguration := "EeMonitorData".machineConfiguration, machineOperation := "EeMonitorData".machineOperation, measConfiguration := "EeMonitorData".measConfiguration, measOperation := "EeMonitorData".measOperation, error => "EeMonitorData".calcError, status => "EeMonitorData".calcStatus)
   END_RUNG
   // the same network as SCL:
   EnS_EEm_Calc(machineConfiguration := "EeMonitorData".machineConfiguration,
                machineOperation := "EeMonitorData".machineOperation,
                measConfiguration := "EeMonitorData".measConfiguration,
                measOperation := "EeMonitorData".measOperation,
                error => "EeMonitorData".calcError,
                status => "EeMonitorData".calcStatus);
END_REGION

REGION Network 5: EE-Monitor: Call EnS_EEm_Report
   // EEm_Report - Write data to MMC
   RUNG wire#powerrail
      "InstEnSeemReport".EnS_EEm_Report(request := "EeMonitorData".reportCreateCsv, machineConfiguration := "EeMonitorData".machineConfiguration, machineOperation := "EeMonitorData".machineOperation, measValueConfiguration := "EeMonitorData".measConfiguration, measValueOperation := "EeMonitorData".measOperation, busy =>, done =>, error =>, status => "EeMonitorData".reportStatus, dataLogNameAct => "EeMonitorData".reportNameCsv)
   END_RUNG
   // the same network as SCL:
   "InstEnSeemReport"(request := "EeMonitorData".reportCreateCsv,   // EnS_EEm_Report
                      machineConfiguration := "EeMonitorData".machineConfiguration,
                      machineOperation := "EeMonitorData".machineOperation,
                      measValueConfiguration := "EeMonitorData".measConfiguration,
                      measValueOperation := "EeMonitorData".measOperation,
                      status => "EeMonitorData".reportStatus,
                      dataLogNameAct => "EeMonitorData".reportNameCsv);
END_REGION
END_FUNCTION

ORGANIZATION_BLOCK "ProgrammingError"   // OB121, LAD, ProgrammingError
// stored: SetENOAutomatically false
   VAR_INPUT
      BlockNr : UInt;   // Number of causing block
      Reaction : USInt;   // 0:ignore, 1:substitute, 2:skip
      Fault_ID : Byte;   // Fault identifier
      BlockType : USInt;   // 16#01:OB, 16#02:FC, 16#03:FB, 16#04:SFC, 16#05:SFB, 16#06:DB: Type of block causing the error
      Area : USInt;   // Area where the error occured
      DBNr : DB_ANY;   // DB number if Area = DB or DI
      Csg_OBNr : OB_ANY;   // Number of OB causing the error
      Csg_Prio : USInt;   // Priority of OB causing the error
      Width : USInt;   // 0:bit, 1:byte, 2:word, 3:dword, 4:lword
   END_VAR
BEGIN
END_ORGANIZATION_BLOCK

ORGANIZATION_BLOCK "Startup"   // OB100, LAD, Startup
TITLE = "Complete Restart"
// stored: AutoNumber false, IsIECCheckEnabled true, SetENOAutomatically true
   VAR_INPUT
      LostRetentive : Bool;   // True if retentive data are lost
      LostRTC : Bool;   // True if date and time are lost
   END_VAR
   VAR_TEMP
      tempError : Bool;
      tempStatus : Word;
      tempDiagnostics : "LAF_typeDiagnosticsSimple";
   END_VAR
BEGIN

REGION Network 1: Set first cycle bit
   // Set the first cycle signal
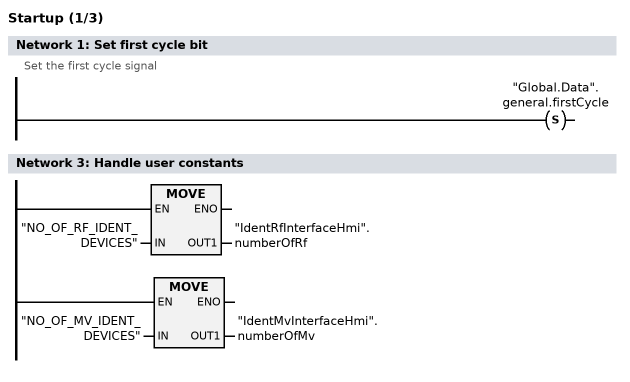
   RUNG wire#powerrail
      S_Coil( "Global.Data".general.firstCycle )
   END_RUNG
   // the same network as SCL:
   "Global.Data".general.firstCycle := TRUE;
END_REGION

REGION Network 2: Enable global power
   // Set global power to true by default. This can be adjusted depending on the user requirement for a specific machine.
END_REGION

REGION Network 3: Handle user constants
   RUNG wire#powerrail
      Move(in := "NO_OF_RF_IDENT_DEVICES", out1 => "IdentRfInterfaceHmi".numberOfRf)
   END_RUNG
   RUNG wire#powerrail
      Move(in := "NO_OF_MV_IDENT_DEVICES", out1 => "IdentMvInterfaceHmi".numberOfMv)
   END_RUNG
   // the same network as SCL:
   "IdentRfInterfaceHmi".numberOfRf := "NO_OF_RF_IDENT_DEVICES";
   "IdentMvInterfaceHmi".numberOfMv := "NO_OF_MV_IDENT_DEVICES";
END_REGION

REGION Network 4: Set drive objects for drive diagnostic
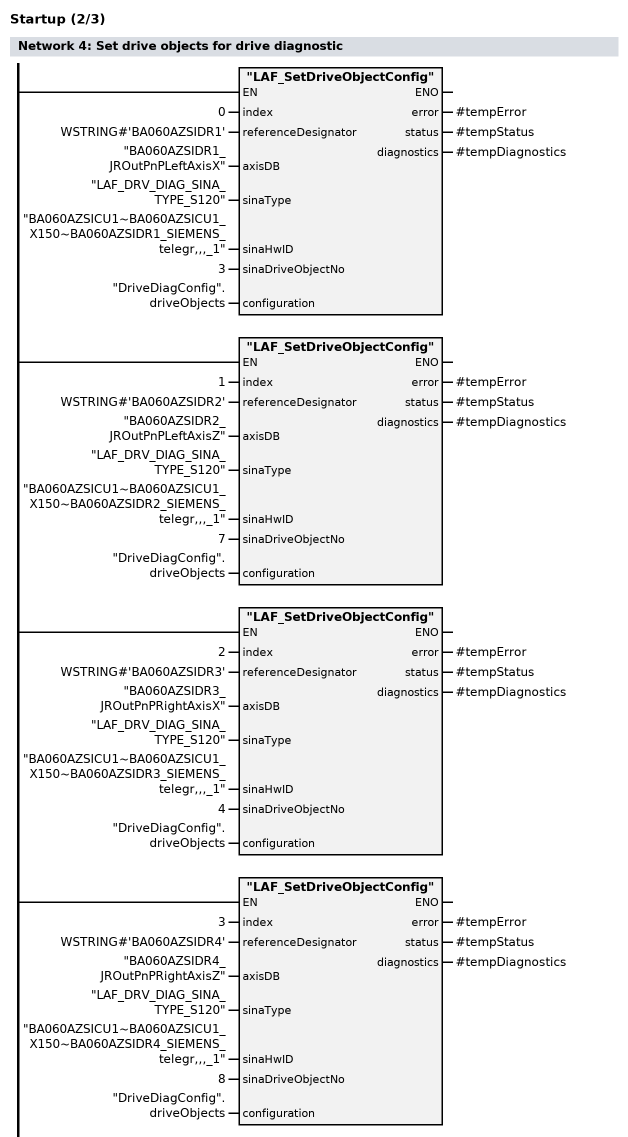
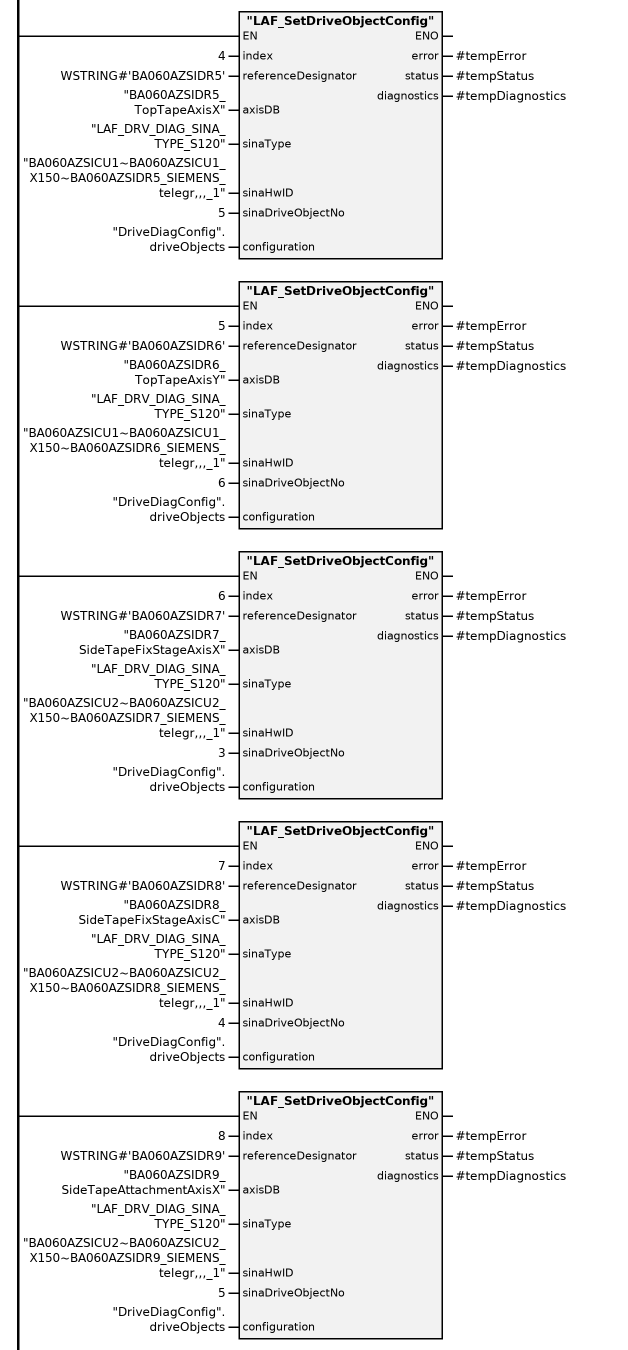
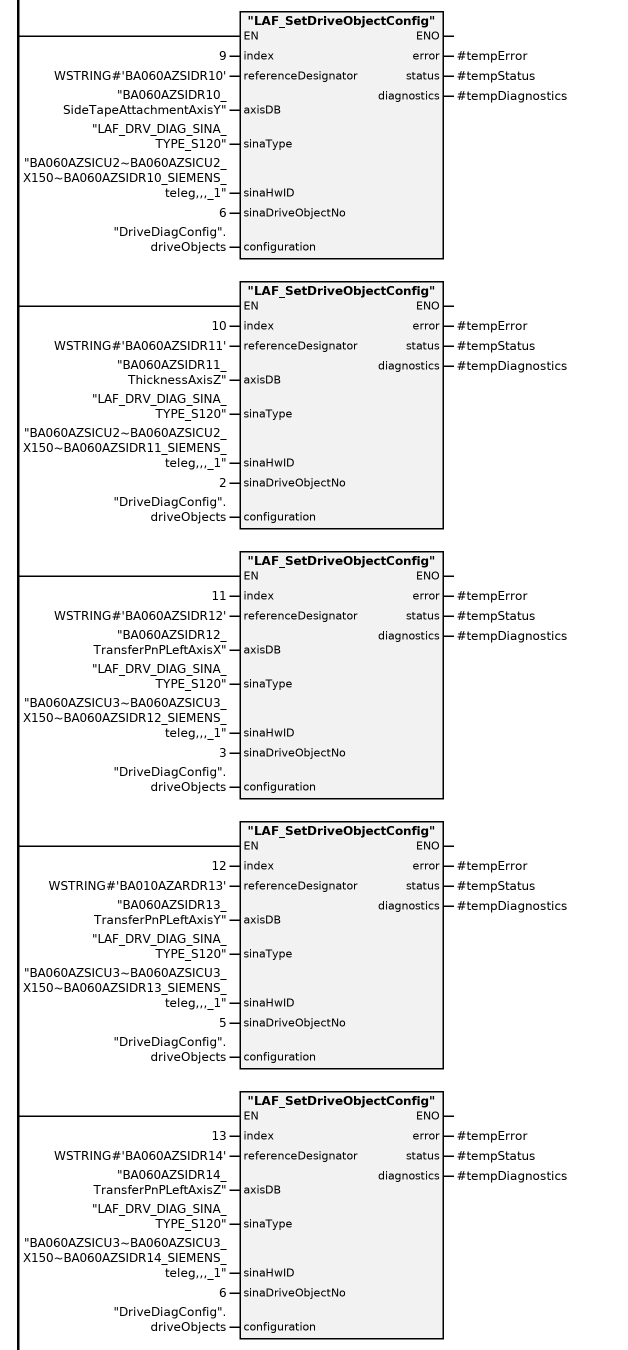
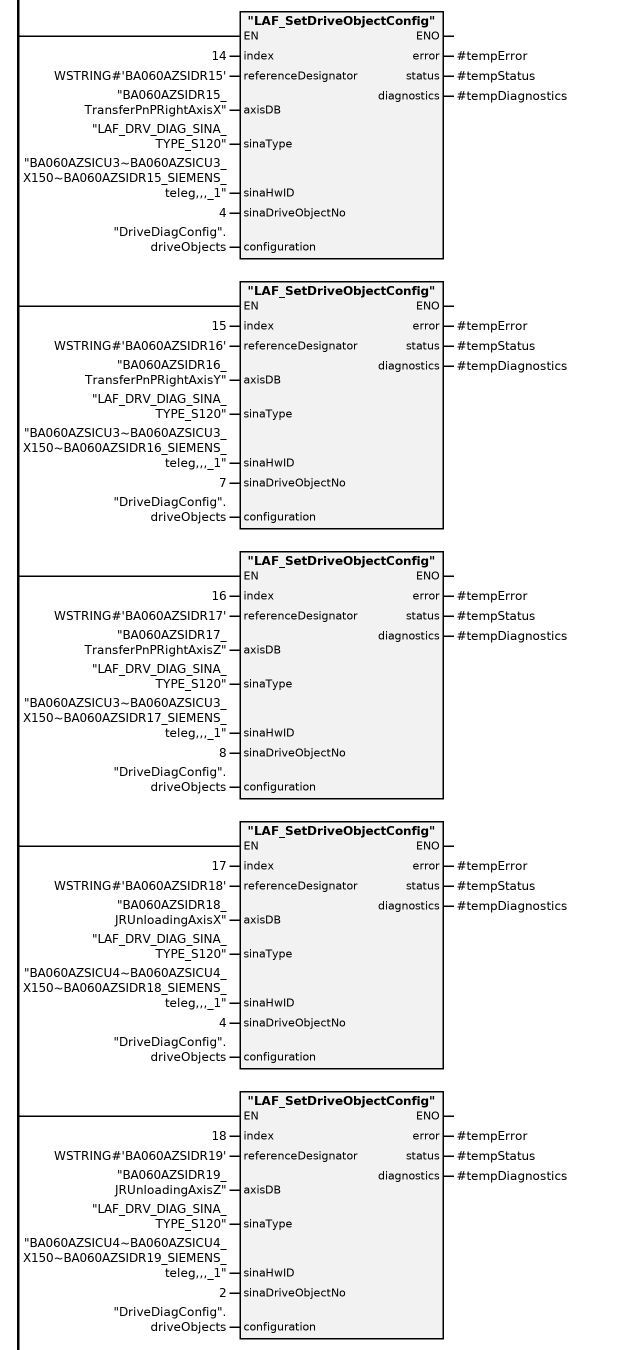
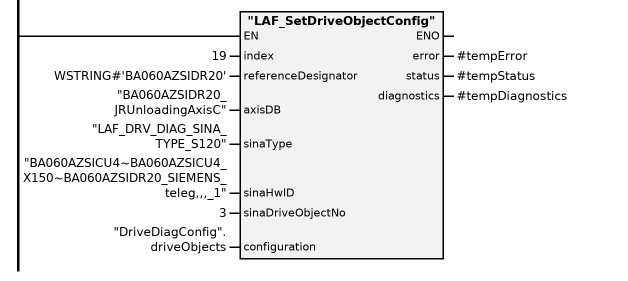
   RUNG wire#powerrail
      "LAF_SetDriveObjectConfig"(index := 0, referenceDesignator := WSTRING#'BA060AZSIDR1', axisDB := "BA060AZSIDR1_JROutPnPLeftAxisX", sinaType := "LAF_DRV_DIAG_SINA_TYPE_S120", sinaHwID := "BA060AZSICU1~BA060AZSICU1_X150~BA060AZSIDR1_SIEMENS_telegr,,,_1", sinaDriveObjectNo := 3, configuration := "DriveDiagConfig".driveObjects, error => #tempError, status => #tempStatus, diagnostics => #tempDiagnostics)
   END_RUNG
   RUNG wire#powerrail
      "LAF_SetDriveObjectConfig"(index := 1, referenceDesignator := WSTRING#'BA060AZSIDR2', axisDB := "BA060AZSIDR2_JROutPnPLeftAxisZ", sinaType := "LAF_DRV_DIAG_SINA_TYPE_S120", sinaHwID := "BA060AZSICU1~BA060AZSICU1_X150~BA060AZSIDR2_SIEMENS_telegr,,,_1", sinaDriveObjectNo := 7, configuration := "DriveDiagConfig".driveObjects, error => #tempError, status => #tempStatus, diagnostics => #tempDiagnostics)
   END_RUNG
   RUNG wire#powerrail
      "LAF_SetDriveObjectConfig"(index := 2, referenceDesignator := WSTRING#'BA060AZSIDR3', axisDB := "BA060AZSIDR3_JROutPnPRightAxisX", sinaType := "LAF_DRV_DIAG_SINA_TYPE_S120", sinaHwID := "BA060AZSICU1~BA060AZSICU1_X150~BA060AZSIDR3_SIEMENS_telegr,,,_1", sinaDriveObjectNo := 4, configuration := "DriveDiagConfig".driveObjects, error => #tempError, status => #tempStatus, diagnostics => #tempDiagnostics)
   END_RUNG
   RUNG wire#powerrail
      "LAF_SetDriveObjectConfig"(index := 3, referenceDesignator := WSTRING#'BA060AZSIDR4', axisDB := "BA060AZSIDR4_JROutPnPRightAxisZ", sinaType := "LAF_DRV_DIAG_SINA_TYPE_S120", sinaHwID := "BA060AZSICU1~BA060AZSICU1_X150~BA060AZSIDR4_SIEMENS_telegr,,,_1", sinaDriveObjectNo := 8, configuration := "DriveDiagConfig".driveObjects, error => #tempError, status => #tempStatus, diagnostics => #tempDiagnostics)
   END_RUNG
   RUNG wire#powerrail
      "LAF_SetDriveObjectConfig"(index := 4, referenceDesignator := WSTRING#'BA060AZSIDR5', axisDB := "BA060AZSIDR5_TopTapeAxisX", sinaType := "LAF_DRV_DIAG_SINA_TYPE_S120", sinaHwID := "BA060AZSICU1~BA060AZSICU1_X150~BA060AZSIDR5_SIEMENS_telegr,,,_1", sinaDriveObjectNo := 5, configuration := "DriveDiagConfig".driveObjects, error => #tempError, status => #tempStatus, diagnostics => #tempDiagnostics)
   END_RUNG
   RUNG wire#powerrail
      "LAF_SetDriveObjectConfig"(index := 5, referenceDesignator := WSTRING#'BA060AZSIDR6', axisDB := "BA060AZSIDR6_TopTapeAxisY", sinaType := "LAF_DRV_DIAG_SINA_TYPE_S120", sinaHwID := "BA060AZSICU1~BA060AZSICU1_X150~BA060AZSIDR6_SIEMENS_telegr,,,_1", sinaDriveObjectNo := 6, configuration := "DriveDiagConfig".driveObjects, error => #tempError, status => #tempStatus, diagnostics => #tempDiagnostics)
   END_RUNG
   RUNG wire#powerrail
      "LAF_SetDriveObjectConfig"(index := 6, referenceDesignator := WSTRING#'BA060AZSIDR7', axisDB := "BA060AZSIDR7_SideTapeFixStageAxisX", sinaType := "LAF_DRV_DIAG_SINA_TYPE_S120", sinaHwID := "BA060AZSICU2~BA060AZSICU2_X150~BA060AZSIDR7_SIEMENS_telegr,,,_1", sinaDriveObjectNo := 3, configuration := "DriveDiagConfig".driveObjects, error => #tempError, status => #tempStatus, diagnostics => #tempDiagnostics)
   END_RUNG
   RUNG wire#powerrail
      "LAF_SetDriveObjectConfig"(index := 7, referenceDesignator := WSTRING#'BA060AZSIDR8', axisDB := "BA060AZSIDR8_SideTapeFixStageAxisC", sinaType := "LAF_DRV_DIAG_SINA_TYPE_S120", sinaHwID := "BA060AZSICU2~BA060AZSICU2_X150~BA060AZSIDR8_SIEMENS_telegr,,,_1", sinaDriveObjectNo := 4, configuration := "DriveDiagConfig".driveObjects, error => #tempError, status => #tempStatus, diagnostics => #tempDiagnostics)
   END_RUNG
   RUNG wire#powerrail
      "LAF_SetDriveObjectConfig"(index := 8, referenceDesignator := WSTRING#'BA060AZSIDR9', axisDB := "BA060AZSIDR9_SideTapeAttachmentAxisX", sinaType := "LAF_DRV_DIAG_SINA_TYPE_S120", sinaHwID := "BA060AZSICU2~BA060AZSICU2_X150~BA060AZSIDR9_SIEMENS_telegr,,,_1", sinaDriveObjectNo := 5, configuration := "DriveDiagConfig".driveObjects, error => #tempError, status => #tempStatus, diagnostics => #tempDiagnostics)
   END_RUNG
   RUNG wire#powerrail
      "LAF_SetDriveObjectConfig"(index := 9, referenceDesignator := WSTRING#'BA060AZSIDR10', axisDB := "BA060AZSIDR10_SideTapeAttachmentAxisY", sinaType := "LAF_DRV_DIAG_SINA_TYPE_S120", sinaHwID := "BA060AZSICU2~BA060AZSICU2_X150~BA060AZSIDR10_SIEMENS_teleg,,,_1", sinaDriveObjectNo := 6, configuration := "DriveDiagConfig".driveObjects, error => #tempError, status => #tempStatus, diagnostics => #tempDiagnostics)
   END_RUNG
   RUNG wire#powerrail
      "LAF_SetDriveObjectConfig"(index := 10, referenceDesignator := WSTRING#'BA060AZSIDR11', axisDB := "BA060AZSIDR11_ThicknessAxisZ", sinaType := "LAF_DRV_DIAG_SINA_TYPE_S120", sinaHwID := "BA060AZSICU2~BA060AZSICU2_X150~BA060AZSIDR11_SIEMENS_teleg,,,_1", sinaDriveObjectNo := 2, configuration := "DriveDiagConfig".driveObjects, error => #tempError, status => #tempStatus, diagnostics => #tempDiagnostics)
   END_RUNG
   RUNG wire#powerrail
      "LAF_SetDriveObjectConfig"(index := 11, referenceDesignator := WSTRING#'BA060AZSIDR12', axisDB := "BA060AZSIDR12_TransferPnPLeftAxisX", sinaType := "LAF_DRV_DIAG_SINA_TYPE_S120", sinaHwID := "BA060AZSICU3~BA060AZSICU3_X150~BA060AZSIDR12_SIEMENS_teleg,,,_1", sinaDriveObjectNo := 3, configuration := "DriveDiagConfig".driveObjects, error => #tempError, status => #tempStatus, diagnostics => #tempDiagnostics)
   END_RUNG
   RUNG wire#powerrail
      "LAF_SetDriveObjectConfig"(index := 12, referenceDesignator := WSTRING#'BA010AZARDR13', axisDB := "BA060AZSIDR13_TransferPnPLeftAxisY", sinaType := "LAF_DRV_DIAG_SINA_TYPE_S120", sinaHwID := "BA060AZSICU3~BA060AZSICU3_X150~BA060AZSIDR13_SIEMENS_teleg,,,_1", sinaDriveObjectNo := 5, configuration := "DriveDiagConfig".driveObjects, error => #tempError, status => #tempStatus, diagnostics => #tempDiagnostics)
   END_RUNG
   RUNG wire#powerrail
      "LAF_SetDriveObjectConfig"(index := 13, referenceDesignator := WSTRING#'BA060AZSIDR14', axisDB := "BA060AZSIDR14_TransferPnPLeftAxisZ", sinaType := "LAF_DRV_DIAG_SINA_TYPE_S120", sinaHwID := "BA060AZSICU3~BA060AZSICU3_X150~BA060AZSIDR14_SIEMENS_teleg,,,_1", sinaDriveObjectNo := 6, configuration := "DriveDiagConfig".driveObjects, error => #tempError, status => #tempStatus, diagnostics => #tempDiagnostics)
   END_RUNG
   RUNG wire#powerrail
      "LAF_SetDriveObjectConfig"(index := 14, referenceDesignator := WSTRING#'BA060AZSIDR15', axisDB := "BA060AZSIDR15_TransferPnPRightAxisX", sinaType := "LAF_DRV_DIAG_SINA_TYPE_S120", sinaHwID := "BA060AZSICU3~BA060AZSICU3_X150~BA060AZSIDR15_SIEMENS_teleg,,,_1", sinaDriveObjectNo := 4, configuration := "DriveDiagConfig".driveObjects, error => #tempError, status => #tempStatus, diagnostics => #tempDiagnostics)
   END_RUNG
   RUNG wire#powerrail
      "LAF_SetDriveObjectConfig"(index := 15, referenceDesignator := WSTRING#'BA060AZSIDR16', axisDB := "BA060AZSIDR16_TransferPnPRightAxisY", sinaType := "LAF_DRV_DIAG_SINA_TYPE_S120", sinaHwID := "BA060AZSICU3~BA060AZSICU3_X150~BA060AZSIDR16_SIEMENS_teleg,,,_1", sinaDriveObjectNo := 7, configuration := "DriveDiagConfig".driveObjects, error => #tempError, status => #tempStatus, diagnostics => #tempDiagnostics)
   END_RUNG
   RUNG wire#powerrail
      "LAF_SetDriveObjectConfig"(index := 16, referenceDesignator := WSTRING#'BA060AZSIDR17', axisDB := "BA060AZSIDR17_TransferPnPRightAxisZ", sinaType := "LAF_DRV_DIAG_SINA_TYPE_S120", sinaHwID := "BA060AZSICU3~BA060AZSICU3_X150~BA060AZSIDR17_SIEMENS_teleg,,,_1", sinaDriveObjectNo := 8, configuration := "DriveDiagConfig".driveObjects, error => #tempError, status => #tempStatus, diagnostics => #tempDiagnostics)
   END_RUNG
   RUNG wire#powerrail
      "LAF_SetDriveObjectConfig"(index := 17, referenceDesignator := WSTRING#'BA060AZSIDR18', axisDB := "BA060AZSIDR18_JRUnloadingAxisX", sinaType := "LAF_DRV_DIAG_SINA_TYPE_S120", sinaHwID := "BA060AZSICU4~BA060AZSICU4_X150~BA060AZSIDR18_SIEMENS_teleg,,,_1", sinaDriveObjectNo := 4, configuration := "DriveDiagConfig".driveObjects, error => #tempError, status => #tempStatus, diagnostics => #tempDiagnostics)
   END_RUNG
   RUNG wire#powerrail
      "LAF_SetDriveObjectConfig"(index := 18, referenceDesignator := WSTRING#'BA060AZSIDR19', axisDB := "BA060AZSIDR19_JRUnloadingAxisZ", sinaType := "LAF_DRV_DIAG_SINA_TYPE_S120", sinaHwID := "BA060AZSICU4~BA060AZSICU4_X150~BA060AZSIDR19_SIEMENS_teleg,,,_1", sinaDriveObjectNo := 2, configuration := "DriveDiagConfig".driveObjects, error => #tempError, status => #tempStatus, diagnostics => #tempDiagnostics)
   END_RUNG
   RUNG wire#powerrail
      "LAF_SetDriveObjectConfig"(index := 19, referenceDesignator := WSTRING#'BA060AZSIDR20', axisDB := "BA060AZSIDR20_JRUnloadingAxisC", sinaType := "LAF_DRV_DIAG_SINA_TYPE_S120", sinaHwID := "BA060AZSICU4~BA060AZSICU4_X150~BA060AZSIDR20_SIEMENS_teleg,,,_1", sinaDriveObjectNo := 3, configuration := "DriveDiagConfig".driveObjects, error => #tempError, status => #tempStatus, diagnostics => #tempDiagnostics)
   END_RUNG
   // the same network as SCL:
   "LAF_SetDriveObjectConfig"(index := 0,
                           referenceDesignator := WSTRING#'BA060AZSIDR1',
                           axisDB := "BA060AZSIDR1_JROutPnPLeftAxisX",
                           sinaType := "LAF_DRV_DIAG_SINA_TYPE_S120",
                           sinaHwID := "BA060AZSICU1~BA060AZSICU1_X150~BA060AZSIDR1_SIEMENS_telegr,,,_1",
                           sinaDriveObjectNo := 3,
                           configuration := "DriveDiagConfig".driveObjects,
                           error => #tempError,
                           status => #tempStatus,
                           diagnostics => #tempDiagnostics);
   "LAF_SetDriveObjectConfig"(index := 1,
                           referenceDesignator := WSTRING#'BA060AZSIDR2',
                           axisDB := "BA060AZSIDR2_JROutPnPLeftAxisZ",
                           sinaType := "LAF_DRV_DIAG_SINA_TYPE_S120",
                           sinaHwID := "BA060AZSICU1~BA060AZSICU1_X150~BA060AZSIDR2_SIEMENS_telegr,,,_1",
                           sinaDriveObjectNo := 7,
                           configuration := "DriveDiagConfig".driveObjects,
                           error => #tempError,
                           status => #tempStatus,
                           diagnostics => #tempDiagnostics);
   "LAF_SetDriveObjectConfig"(index := 2,
                           referenceDesignator := WSTRING#'BA060AZSIDR3',
                           axisDB := "BA060AZSIDR3_JROutPnPRightAxisX",
                           sinaType := "LAF_DRV_DIAG_SINA_TYPE_S120",
                           sinaHwID := "BA060AZSICU1~BA060AZSICU1_X150~BA060AZSIDR3_SIEMENS_telegr,,,_1",
                           sinaDriveObjectNo := 4,
                           configuration := "DriveDiagConfig".driveObjects,
                           error => #tempError,
                           status => #tempStatus,
                           diagnostics => #tempDiagnostics);
   "LAF_SetDriveObjectConfig"(index := 3,
                           referenceDesignator := WSTRING#'BA060AZSIDR4',
                           axisDB := "BA060AZSIDR4_JROutPnPRightAxisZ",
                           sinaType := "LAF_DRV_DIAG_SINA_TYPE_S120",
                           sinaHwID := "BA060AZSICU1~BA060AZSICU1_X150~BA060AZSIDR4_SIEMENS_telegr,,,_1",
                           sinaDriveObjectNo := 8,
                           configuration := "DriveDiagConfig".driveObjects,
                           error => #tempError,
                           status => #tempStatus,
                           diagnostics => #tempDiagnostics);
   "LAF_SetDriveObjectConfig"(index := 4,
                           referenceDesignator := WSTRING#'BA060AZSIDR5',
                           axisDB := "BA060AZSIDR5_TopTapeAxisX",
                           sinaType := "LAF_DRV_DIAG_SINA_TYPE_S120",
                           sinaHwID := "BA060AZSICU1~BA060AZSICU1_X150~BA060AZSIDR5_SIEMENS_telegr,,,_1",
                           sinaDriveObjectNo := 5,
                           configuration := "DriveDiagConfig".driveObjects,
                           error => #tempError,
                           status => #tempStatus,
                           diagnostics => #tempDiagnostics);
   "LAF_SetDriveObjectConfig"(index := 5,
                           referenceDesignator := WSTRING#'BA060AZSIDR6',
                           axisDB := "BA060AZSIDR6_TopTapeAxisY",
                           sinaType := "LAF_DRV_DIAG_SINA_TYPE_S120",
                           sinaHwID := "BA060AZSICU1~BA060AZSICU1_X150~BA060AZSIDR6_SIEMENS_telegr,,,_1",
                           sinaDriveObjectNo := 6,
                           configuration := "DriveDiagConfig".driveObjects,
                           error => #tempError,
                           status => #tempStatus,
                           diagnostics => #tempDiagnostics);
   "LAF_SetDriveObjectConfig"(index := 6,
                           referenceDesignator := WSTRING#'BA060AZSIDR7',
                           axisDB := "BA060AZSIDR7_SideTapeFixStageAxisX",
                           sinaType := "LAF_DRV_DIAG_SINA_TYPE_S120",
                           sinaHwID := "BA060AZSICU2~BA060AZSICU2_X150~BA060AZSIDR7_SIEMENS_telegr,,,_1",
                           sinaDriveObjectNo := 3,
                           configuration := "DriveDiagConfig".driveObjects,
                           error => #tempError,
                           status => #tempStatus,
                           diagnostics => #tempDiagnostics);
   "LAF_SetDriveObjectConfig"(index := 7,
                           referenceDesignator := WSTRING#'BA060AZSIDR8',
                           axisDB := "BA060AZSIDR8_SideTapeFixStageAxisC",
                           sinaType := "LAF_DRV_DIAG_SINA_TYPE_S120",
                           sinaHwID := "BA060AZSICU2~BA060AZSICU2_X150~BA060AZSIDR8_SIEMENS_telegr,,,_1",
                           sinaDriveObjectNo := 4,
                           configuration := "DriveDiagConfig".driveObjects,
                           error => #tempError,
                           status => #tempStatus,
                           diagnostics => #tempDiagnostics);
   "LAF_SetDriveObjectConfig"(index := 8,
                           referenceDesignator := WSTRING#'BA060AZSIDR9',
                           axisDB := "BA060AZSIDR9_SideTapeAttachmentAxisX",
                           sinaType := "LAF_DRV_DIAG_SINA_TYPE_S120",
                           sinaHwID := "BA060AZSICU2~BA060AZSICU2_X150~BA060AZSIDR9_SIEMENS_telegr,,,_1",
                           sinaDriveObjectNo := 5,
                           configuration := "DriveDiagConfig".driveObjects,
                           error => #tempError,
                           status => #tempStatus,
                           diagnostics => #tempDiagnostics);
   "LAF_SetDriveObjectConfig"(index := 9,
                           referenceDesignator := WSTRING#'BA060AZSIDR10',
                           axisDB := "BA060AZSIDR10_SideTapeAttachmentAxisY",
                           sinaType := "LAF_DRV_DIAG_SINA_TYPE_S120",
                           sinaHwID := "BA060AZSICU2~BA060AZSICU2_X150~BA060AZSIDR10_SIEMENS_teleg,,,_1",
                           sinaDriveObjectNo := 6,
                           configuration := "DriveDiagConfig".driveObjects,
                           error => #tempError,
                           status => #tempStatus,
                           diagnostics => #tempDiagnostics);
   "LAF_SetDriveObjectConfig"(index := 10,
                           referenceDesignator := WSTRING#'BA060AZSIDR11',
                           axisDB := "BA060AZSIDR11_ThicknessAxisZ",
                           sinaType := "LAF_DRV_DIAG_SINA_TYPE_S120",
                           sinaHwID := "BA060AZSICU2~BA060AZSICU2_X150~BA060AZSIDR11_SIEMENS_teleg,,,_1",
                           sinaDriveObjectNo := 2,
                           configuration := "DriveDiagConfig".driveObjects,
                           error => #tempError,
                           status => #tempStatus,
                           diagnostics => #tempDiagnostics);
   "LAF_SetDriveObjectConfig"(index := 11,
                           referenceDesignator := WSTRING#'BA060AZSIDR12',
                           axisDB := "BA060AZSIDR12_TransferPnPLeftAxisX",
                           sinaType := "LAF_DRV_DIAG_SINA_TYPE_S120",
                           sinaHwID := "BA060AZSICU3~BA060AZSICU3_X150~BA060AZSIDR12_SIEMENS_teleg,,,_1",
                           sinaDriveObjectNo := 3,
                           configuration := "DriveDiagConfig".driveObjects,
                           error => #tempError,
                           status => #tempStatus,
                           diagnostics => #tempDiagnostics);
   "LAF_SetDriveObjectConfig"(index := 12,
                           referenceDesignator := WSTRING#'BA010AZARDR13',
                           axisDB := "BA060AZSIDR13_TransferPnPLeftAxisY",
                           sinaType := "LAF_DRV_DIAG_SINA_TYPE_S120",
                           sinaHwID := "BA060AZSICU3~BA060AZSICU3_X150~BA060AZSIDR13_SIEMENS_teleg,,,_1",
                           sinaDriveObjectNo := 5,
                           configuration := "DriveDiagConfig".driveObjects,
                           error => #tempError,
                           status => #tempStatus,
                           diagnostics => #tempDiagnostics);
   "LAF_SetDriveObjectConfig"(index := 13,
                           referenceDesignator := WSTRING#'BA060AZSIDR14',
                           axisDB := "BA060AZSIDR14_TransferPnPLeftAxisZ",
                           sinaType := "LAF_DRV_DIAG_SINA_TYPE_S120",
                           sinaHwID := "BA060AZSICU3~BA060AZSICU3_X150~BA060AZSIDR14_SIEMENS_teleg,,,_1",
                           sinaDriveObjectNo := 6,
                           configuration := "DriveDiagConfig".driveObjects,
                           error => #tempError,
                           status => #tempStatus,
                           diagnostics => #tempDiagnostics);
   "LAF_SetDriveObjectConfig"(index := 14,
                           referenceDesignator := WSTRING#'BA060AZSIDR15',
                           axisDB := "BA060AZSIDR15_TransferPnPRightAxisX",
                           sinaType := "LAF_DRV_DIAG_SINA_TYPE_S120",
                           sinaHwID := "BA060AZSICU3~BA060AZSICU3_X150~BA060AZSIDR15_SIEMENS_teleg,,,_1",
                           sinaDriveObjectNo := 4,
                           configuration := "DriveDiagConfig".driveObjects,
                           error => #tempError,
                           status => #tempStatus,
                           diagnostics => #tempDiagnostics);
   "LAF_SetDriveObjectConfig"(index := 15,
                           referenceDesignator := WSTRING#'BA060AZSIDR16',
                           axisDB := "BA060AZSIDR16_TransferPnPRightAxisY",
                           sinaType := "LAF_DRV_DIAG_SINA_TYPE_S120",
                           sinaHwID := "BA060AZSICU3~BA060AZSICU3_X150~BA060AZSIDR16_SIEMENS_teleg,,,_1",
                           sinaDriveObjectNo := 7,
                           configuration := "DriveDiagConfig".driveObjects,
                           error => #tempError,
                           status => #tempStatus,
                           diagnostics => #tempDiagnostics);
   "LAF_SetDriveObjectConfig"(index := 16,
                           referenceDesignator := WSTRING#'BA060AZSIDR17',
                           axisDB := "BA060AZSIDR17_TransferPnPRightAxisZ",
                           sinaType := "LAF_DRV_DIAG_SINA_TYPE_S120",
                           sinaHwID := "BA060AZSICU3~BA060AZSICU3_X150~BA060AZSIDR17_SIEMENS_teleg,,,_1",
                           sinaDriveObjectNo := 8,
                           configuration := "DriveDiagConfig".driveObjects,
                           error => #tempError,
                           status => #tempStatus,
                           diagnostics => #tempDiagnostics);
   "LAF_SetDriveObjectConfig"(index := 17,
                           referenceDesignator := WSTRING#'BA060AZSIDR18',
                           axisDB := "BA060AZSIDR18_JRUnloadingAxisX",
                           sinaType := "LAF_DRV_DIAG_SINA_TYPE_S120",
                           sinaHwID := "BA060AZSICU4~BA060AZSICU4_X150~BA060AZSIDR18_SIEMENS_teleg,,,_1",
                           sinaDriveObjectNo := 4,
                           configuration := "DriveDiagConfig".driveObjects,
                           error => #tempError,
                           status => #tempStatus,
                           diagnostics => #tempDiagnostics);
   "LAF_SetDriveObjectConfig"(index := 18,
                           referenceDesignator := WSTRING#'BA060AZSIDR19',
                           axisDB := "BA060AZSIDR19_JRUnloadingAxisZ",
                           sinaType := "LAF_DRV_DIAG_SINA_TYPE_S120",
                           sinaHwID := "BA060AZSICU4~BA060AZSICU4_X150~BA060AZSIDR19_SIEMENS_teleg,,,_1",
                           sinaDriveObjectNo := 2,
                           configuration := "DriveDiagConfig".driveObjects,
                           error => #tempError,
                           status => #tempStatus,
                           diagnostics => #tempDiagnostics);
   "LAF_SetDriveObjectConfig"(index := 19,
                           referenceDesignator := WSTRING#'BA060AZSIDR20',
                           axisDB := "BA060AZSIDR20_JRUnloadingAxisC",
                           sinaType := "LAF_DRV_DIAG_SINA_TYPE_S120",
                           sinaHwID := "BA060AZSICU4~BA060AZSICU4_X150~BA060AZSIDR20_SIEMENS_teleg,,,_1",
                           sinaDriveObjectNo := 3,
                           configuration := "DriveDiagConfig".driveObjects,
                           error => #tempError,
                           status => #tempStatus,
                           diagnostics => #tempDiagnostics);
END_REGION

REGION Network 5: Manual Operation Line
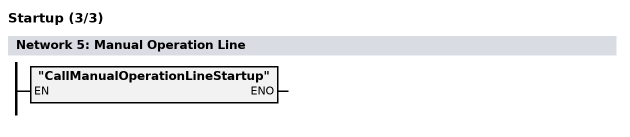
   RUNG wire#powerrail
      "CallManualOperationLineStartup"()
   END_RUNG
   // the same network as SCL:
   "CallManualOperationLineStartup"();
END_REGION

REGION Network 6 (SCL): Configuration Set Position
   //DR01
   "Unit1.Em2.HmiInterface".cmJROutPnPLeftAxisX.configuration.setPositions := "AxisDataBackUp_DB".DR1."configuration.setPositions";
   //Unit1.Em2.HmiInterface.cm.softcam.jrOutPnPLeftAxisX := "AxisDataBackUp_DB".DR1.softcam;


   //DR02
   "Unit1.Em2.HmiInterface".cmJROutPnPLeftAxisZ.configuration.setPositions := "AxisDataBackUp_DB".DR2."configuration.setPositions";
   //Unit1.Em2.HmiInterface.cm.softcam.jrOutPnPLeftAxisZ := "AxisDataBackUp_DB".DR2.softcam;


   //DR03
   "Unit1.Em2.HmiInterface".cmJROutPnPRightAxisX.configuration.setPositions := "AxisDataBackUp_DB".DR3."configuration.setPositions";
   //Unit1.Em2.HmiInterface.cm.softcam.jrOutPnPRightAxisX := "AxisDataBackUp_DB".DR3.softcam;


   //DR04
   "Unit1.Em2.HmiInterface".cmJROutPnPRightAxisZ.configuration.setPositions := "AxisDataBackUp_DB".DR4."configuration.setPositions";
   //Unit1.Em2.HmiInterface.cm.softcam.jrOutPnPRightAxisZ := "AxisDataBackUp_DB".DR4.softcam;


   //DR05
   "Unit1.Em3.HmiInterface".cmTopTapeAxisX.configuration.setPositions := "AxisDataBackUp_DB".DR5."configuration.setPositions";
   //Unit1.Em3.HmiInterface.cm.softcam.topTapeAxisX := "AxisDataBackUp_DB".DR5.softcam;


   //DR06
   "Unit1.Em3.HmiInterface".cmTopTapeAxisY.configuration.setPositions := "AxisDataBackUp_DB".DR6."configuration.setPositions";
   //Unit1.Em3.HmiInterface.cm.softcam.topTapeAxisY := "AxisDataBackUp_DB".DR6.softcam;


   //DR07
   "Unit1.Em4.HmiInterface".cmSideTapeFixStageAxisX.configuration.setPositions := "AxisDataBackUp_DB".DR7."configuration.setPositions";
   //Unit1.Em4.HmiInterface.cm.softcam.sideTapeFixStageAxisX := "AxisDataBackUp_DB".DR7.softcam;


   //DR08
   "Unit1.Em4.HmiInterface".cmSideTapeFixStageAxisC.configuration.setPositions := "AxisDataBackUp_DB".DR8."configuration.setPositions";
   //Unit1.Em4.HmiInterface.cm.softcam.sideTapeFixStageAxisC := "AxisDataBackUp_DB".DR8.softcam;


   //DR09
   "Unit1.Em4.HmiInterface".cmSideTapeAttachmentAxisX.configuration.setPositions := "AxisDataBackUp_DB".DR9."configuration.setPositions";
   //Unit1.Em4.HmiInterface.cm.softcam.sideTapeAttachmentAxisX := "AxisDataBackUp_DB".DR9.softcam;


   //DR10
   "Unit1.Em4.HmiInterface".cmSideTapeAttachmentAxisY.configuration.setPositions := "AxisDataBackUp_DB".DR10."configuration.setPositions";
   //Unit1.Em4.HmiInterface.cm.softcam.sideTapeAttachmentAxisY := "AxisDataBackUp_DB".DR10.softcam;


   //DR11
   "Unit1.Em8.HmiInterface".cmThicknessAxisZ.configuration.setPositions := "AxisDataBackUp_DB".DR11."configuration.setPositions";
   //Unit1.Em8.HmiInterface.cm.softcam.thicknessAxisZ := "AxisDataBackUp_DB".DR11.softcam;


   //DR12
   "Unit1.Em5.HmiInterface".cmTransferPnPLeftAxisX.configuration.setPositions := "AxisDataBackUp_DB".DR12."configuration.setPositions";
   //Unit1.Em5.HmiInterface.cm.softcam.transferPnPLeftAxisX := "AxisDataBackUp_DB".DR12.softcam;

   //DR13
   "Unit1.Em5.HmiInterface".cmTransferPnPLeftAxisY.configuration.setPositions := "AxisDataBackUp_DB".DR13."configuration.setPositions";
   //Unit1.Em5.HmiInterface.cm.softcam.transferPnPLeftAxisY := "AxisDataBackUp_DB".DR13.softcam;


   //DR14
   "Unit1.Em5.HmiInterface".cmTransferPnPLeftAxisZ.configuration.setPositions := "AxisDataBackUp_DB".DR14."configuration.setPositions";
   //Unit1.Em5.HmiInterface.cm.softcam.transferPnPLeftAxisZ := "AxisDataBackUp_DB".DR14.softcam;


   //DR15
   "Unit1.Em5.HmiInterface".cmTransferPnPRightAxisX.configuration.setPositions := "AxisDataBackUp_DB".DR15."configuration.setPositions";
   //Unit1.Em5.HmiInterface.cm.softcam.transferPnPRightAxisX := "AxisDataBackUp_DB".DR15.softcam;


   //DR16
   "Unit1.Em5.HmiInterface".cmTransferPnPRightAxisY.configuration.setPositions := "AxisDataBackUp_DB".DR16."configuration.setPositions";
   //Unit1.Em5.HmiInterface.cm.softcam.transferPnPRightAxisY := "AxisDataBackUp_DB".DR16.softcam;


   //DR17
   "Unit1.Em5.HmiInterface".cmTransferPnPRightAxisZ.configuration.setPositions := "AxisDataBackUp_DB".DR17."configuration.setPositions";
   //Unit1.Em5.HmiInterface.cm.softcam.transferPnPRightAxisZ := "AxisDataBackUp_DB".DR17.softcam;


   //DR18
   "Unit1.Em13.HmiInterface".cmJRUnloadingPnPAxisX.configuration.setPositions := "AxisDataBackUp_DB".DR18."configuration.setPositions";
   //Unit1.Em13.HmiInterface.cm.softcam.jrUnloadingPnPAxisX := "AxisDataBackUp_DB".DR18.softcam;


   //DR19
   "Unit1.Em13.HmiInterface".cmJRUnloadingPnPAxisZ.configuration.setPositions := "AxisDataBackUp_DB".DR19."configuration.setPositions";
   //Unit1.Em13.HmiInterface.cm.softcam.jrUnloadingPnPAxisZ := "AxisDataBackUp_DB".DR19.softcam;


   //DR20
   "Unit1.Em13.HmiInterface".cmJRUnloadingPnPAxisC.configuration.setPositions := "AxisDataBackUp_DB".DR20."configuration.setPositions";
   //Unit1.Em13.HmiInterface.cm.softcam.jrUnloadingPnPAxisC := "AxisDataBackUp_DB".DR20.softcam;
END_REGION
END_ORGANIZATION_BLOCK

FUNCTION "CallManualOperationLineStartup" : Void
{ S7_Optimized_Access := 'TRUE' ; Published := 'FALSE' }
VERSION : 0.1

BEGIN
	REGION Description
	(*
	    Startup call to set the configuration of the Manual Operation Line for the Equipment modules
	*)
	    
	END_REGION
	
	"LAF_InternalManual".emsWithManualOpConfigured.maxNoOfEms := "NO_OF_EM";
	
	REGION Unit 1 Equipment Module 0 configuration
	    "ManualOperationControl_U1Em0".manualOperationEm.equipmentModuleNum := 1010;
	    "ManualOperationControl_U1Em0".manualOperationEmArea[2].displayedLines := '1-;';
	    "ManualOperationControl_U1Em0".manualOperationEmArea[1].displayedLines := '21-27;';
	END_REGION
	
	REGION Unit 1 Equipment Module 1 configuration
	    "ManualOperationControl_U1Em1".manualOperationEm.equipmentModuleNum := 1020;
	    "ManualOperationControl_U1Em1".manualOperationEmArea[2].displayedLines := '1-;';
	    "ManualOperationControl_U1Em1".manualOperationEmArea[1].displayedLines := '21-27;';
	END_REGION
	
	REGION Unit 1 Equipment Module 2 configuration
	    "ManualOperationControl_U1Em2".manualOperationEm.equipmentModuleNum := 1030;
	    "ManualOperationControl_U1Em2".manualOperationEmArea[2].displayedLines := '1-4;';
	    "ManualOperationControl_U1Em2".manualOperationEmArea[1].displayedLines := '21-22;';
	END_REGION
	
	REGION Unit 1 Equipment Module 3 configuration
	    "ManualOperationControl_U1Em3".manualOperationEm.equipmentModuleNum := 1040;
	    "ManualOperationControl_U1Em3".manualOperationEmArea[2].displayedLines := '1-2;';
	    "ManualOperationControl_U1Em3".manualOperationEmArea[1].displayedLines := '21-31;';
	END_REGION
	
	REGION Unit 1 Equipment Module 4 configuration
	    "ManualOperationControl_U1Em4".manualOperationEm.equipmentModuleNum := 1050;
	    "ManualOperationControl_U1Em4".manualOperationEmArea[2].displayedLines := '1-4;';
	    "ManualOperationControl_U1Em4".manualOperationEmArea[1].displayedLines := '21-33;';
	END_REGION
	
	REGION Unit 1 Equipment Module 5 configuration
	    "ManualOperationControl_U1Em5".manualOperationEm.equipmentModuleNum := 1060;
	    "ManualOperationControl_U1Em5".manualOperationEmArea[2].displayedLines := '1-6;';
	    "ManualOperationControl_U1Em5".manualOperationEmArea[1].displayedLines := '21-22;';
	END_REGION
	
	REGION Unit 1 Equipment Module 6 configuration
	    "ManualOperationControl_U1Em6".manualOperationEm.equipmentModuleNum := 1070;
	    "ManualOperationControl_U1Em6".manualOperationEmArea[2].displayedLines := '1;';
	    "ManualOperationControl_U1Em6".manualOperationEmArea[1].displayedLines := '21-24;';
	END_REGION
	
	REGION Unit 1 Equipment Module 7 configuration
	    "ManualOperationControl_U1Em7".manualOperationEm.equipmentModuleNum := 1080;
	    "ManualOperationControl_U1Em7".manualOperationEmArea[2].displayedLines := '1;';
	    "ManualOperationControl_U1Em7".manualOperationEmArea[1].displayedLines := '21-24;';
	END_REGION
	
	 REGION Unit 1 Equipment Module 8 configuration
	     "ManualOperationControl_U1Em8".manualOperationEm.equipmentModuleNum := 1090;
	     "ManualOperationControl_U1Em8".manualOperationEmArea[2].displayedLines := '1-2;';
	     "ManualOperationControl_U1Em8".manualOperationEmArea[1].displayedLines := '21-27;';
	END_REGION
	
	REGION Unit 1 Equipment Module 9 configuration
	    "ManualOperationControl_U1Em9".manualOperationEm.equipmentModuleNum := 1100;
	    "ManualOperationControl_U1Em9".manualOperationEmArea[2].displayedLines := '1-;';
	    "ManualOperationControl_U1Em9".manualOperationEmArea[1].displayedLines := '21-22;';
	END_REGION
	REGION Unit 1 Equipment Module 10 configuration
	    "ManualOperationControl_U1Em10".manualOperationEm.equipmentModuleNum := 1110;
	    "ManualOperationControl_U1Em10".manualOperationEmArea[2].displayedLines := '1-;';
	    "ManualOperationControl_U1Em10".manualOperationEmArea[1].displayedLines := '21-22;';
	END_REGION
	REGION Unit 1 Equipment Module 11 configuration
	    "ManualOperationControl_U1Em11".manualOperationEm.equipmentModuleNum := 1120;
	    "ManualOperationControl_U1Em11".manualOperationEmArea[2].displayedLines := '1-;';
	    "ManualOperationControl_U1Em11".manualOperationEmArea[1].displayedLines := '21-22;';
	END_REGION
	
	REGION Unit 1 Equipment Module 12 configuration
	    "ManualOperationControl_U1Em12".manualOperationEm.equipmentModuleNum := 1130;
	    "ManualOperationControl_U1Em12".manualOperationEmArea[2].displayedLines := '1-;';
	    "ManualOperationControl_U1Em12".manualOperationEmArea[1].displayedLines := '21-27;';
	END_REGION
	
	REGION Unit 1 Equipment Module 13 configuration
	    "ManualOperationControl_U1Em13".manualOperationEm.equipmentModuleNum := 1140;
	    "ManualOperationControl_U1Em13".manualOperationEmArea[2].displayedLines := '1-3;';
	    "ManualOperationControl_U1Em13".manualOperationEmArea[1].displayedLines := '21;';
	END_REGION
	
	(* REGION Unit 1 Equipment Module 14 configuration
	    "ManualOperationControl_U1Em14".manualOperationEm.equipmentModuleNum := 1150;
	    "ManualOperationControl_U1Em14".manualOperationEmArea[2].displayedLines := '1-;';
	    "ManualOperationControl_U1Em14".manualOperationEmArea[1].displayedLines := '13-18;';
	END_REGION
	
	REGION Unit 1 Equipment Module 15 configuration
	    "ManualOperationControl_U1Em15".manualOperationEm.equipmentModuleNum := 1160;
	    "ManualOperationControl_U1Em15".manualOperationEmArea[2].displayedLines := '1-;';
	    "ManualOperationControl_U1Em15".manualOperationEmArea[1].displayedLines := '13-18;';
	END_REGION 
	*)
END_FUNCTION

FUNCTION "LAF_ManualOperationLine_Notes" : Void   // FC23, LAD
TITLE = LAF_ManualOperationLine_Notes
// Here are some points that are important for the use and configuration of manual operation lines:
// 
// * For the appearance of each Line, Json files with the configurations need to be added manually to the target machine. Be it in a PC Runtime or Panel. The Path is set in the HMI as the HMI Tag "manualOperationFilePath" in the "03_manualOperation" table. We have set it to "D:\\JsonFiles\\". The files used for this example are saved in the project UserFiles. The Path for the Panel can look like "/home/industrial/JsonFiles".
// 
// * Under "CallManualOperationLines" are the calls for the main configuration of a Equipment module and the control of each line.
//  * Each Equipment module needs to have a defined number. For the numeration we recommend using the second and third digit for the Equipment module number used in the project and the fourth digit with the number of the unit.
// 
// * The texts for the Areas are defined as text lists in the HMI. For the corresponding group, the naming is currently set as "EquipmentAreas_XXXX" with the XXXX as the Equipment Module number. It is set in the "manualOperationEm.equipmentModuleNum".
//  
// * There can be defined 16 color text lists. Each text list defines: "1 - normal, 2 - pressed, 3 - confirmed, 4 - deactivated, 5 - deactivated+pressed".
//  * The color value is in hex with the 2 first values on the left defining the transparency and the rest as normal color values.
//  * The text list name is currently "LAF_manualColorX" with the X as the text list number.
// 
// * If another HMI device is added, please don't forget the Scheduled tasks for updating the lines  
// 
// * The amount of areas is defined by the size of the array in the configuration of areas. The array should start.
// stored: SetENOAutomatically false
BEGIN
END_FUNCTION

FUNCTION "CallCycleTimerMapping" : Void   // FC32781, LAD
// stored: SetENOAutomatically false
   VAR CONSTANT
      TRUE : Bool := TRUE;
   END_VAR
BEGIN

REGION Network 1: cycleTimerDataSet[1]
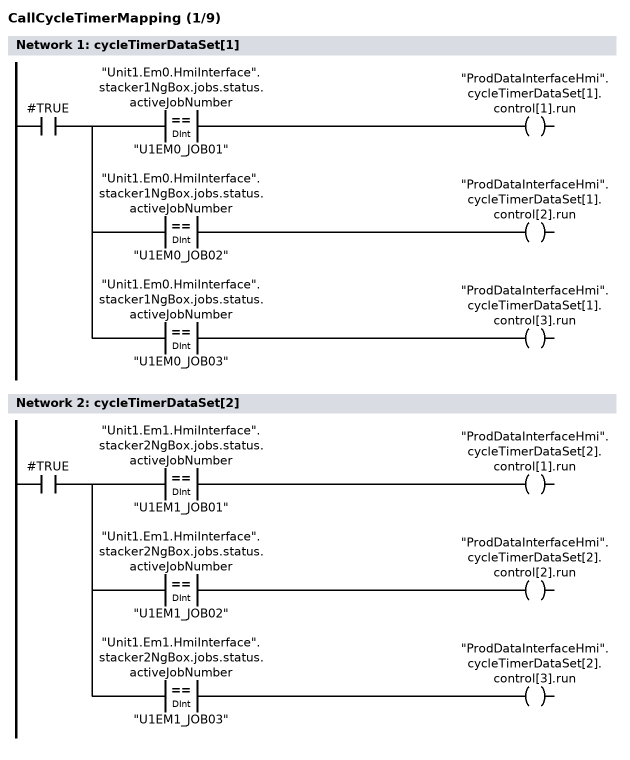
   RUNG wire#powerrail
      Contact( #TRUE )
      wire#w1
      { S7_Templates := "SrcType := DInt" } EQ_Contact(in1 := "Unit1.Em0.HmiInterface".stacker1NgBox.jobs.status.activeJobNumber, in2 := "U1EM0_JOB01")
      Coil( "ProdDataInterfaceHmi".cycleTimerDataSet[1].control[1].run )
   END_RUNG
   RUNG wire#w1
      { S7_Templates := "SrcType := DInt" } EQ_Contact(in1 := "Unit1.Em0.HmiInterface".stacker1NgBox.jobs.status.activeJobNumber, in2 := "U1EM0_JOB02")
      Coil( "ProdDataInterfaceHmi".cycleTimerDataSet[1].control[2].run )
   END_RUNG
   RUNG wire#w1
      { S7_Templates := "SrcType := DInt" } EQ_Contact(in1 := "Unit1.Em0.HmiInterface".stacker1NgBox.jobs.status.activeJobNumber, in2 := "U1EM0_JOB03")
      Coil( "ProdDataInterfaceHmi".cycleTimerDataSet[1].control[3].run )
   END_RUNG
   // the same network as SCL:
   "ProdDataInterfaceHmi".cycleTimerDataSet[1].control[1].run := #TRUE AND ("Unit1.Em0.HmiInterface".stacker1NgBox.jobs.status.activeJobNumber = "U1EM0_JOB01");
   "ProdDataInterfaceHmi".cycleTimerDataSet[1].control[2].run := #TRUE AND ("Unit1.Em0.HmiInterface".stacker1NgBox.jobs.status.activeJobNumber = "U1EM0_JOB02");
   "ProdDataInterfaceHmi".cycleTimerDataSet[1].control[3].run := #TRUE AND ("Unit1.Em0.HmiInterface".stacker1NgBox.jobs.status.activeJobNumber = "U1EM0_JOB03");
END_REGION

REGION Network 2: cycleTimerDataSet[2]
   RUNG wire#powerrail
      Contact( #TRUE )
      wire#w1
      { S7_Templates := "SrcType := DInt" } EQ_Contact(in1 := "Unit1.Em1.HmiInterface".stacker2NgBox.jobs.status.activeJobNumber, in2 := "U1EM1_JOB01")
      Coil( "ProdDataInterfaceHmi".cycleTimerDataSet[2].control[1].run )
   END_RUNG
   RUNG wire#w1
      { S7_Templates := "SrcType := DInt" } EQ_Contact(in1 := "Unit1.Em1.HmiInterface".stacker2NgBox.jobs.status.activeJobNumber, in2 := "U1EM1_JOB02")
      Coil( "ProdDataInterfaceHmi".cycleTimerDataSet[2].control[2].run )
   END_RUNG
   RUNG wire#w1
      { S7_Templates := "SrcType := DInt" } EQ_Contact(in1 := "Unit1.Em1.HmiInterface".stacker2NgBox.jobs.status.activeJobNumber, in2 := "U1EM1_JOB03")
      Coil( "ProdDataInterfaceHmi".cycleTimerDataSet[2].control[3].run )
   END_RUNG
   // the same network as SCL:
   "ProdDataInterfaceHmi".cycleTimerDataSet[2].control[1].run := #TRUE AND ("Unit1.Em1.HmiInterface".stacker2NgBox.jobs.status.activeJobNumber = "U1EM1_JOB01");
   "ProdDataInterfaceHmi".cycleTimerDataSet[2].control[2].run := #TRUE AND ("Unit1.Em1.HmiInterface".stacker2NgBox.jobs.status.activeJobNumber = "U1EM1_JOB02");
   "ProdDataInterfaceHmi".cycleTimerDataSet[2].control[3].run := #TRUE AND ("Unit1.Em1.HmiInterface".stacker2NgBox.jobs.status.activeJobNumber = "U1EM1_JOB03");
END_REGION

REGION Network 3: cycleTimerDataSet[3]
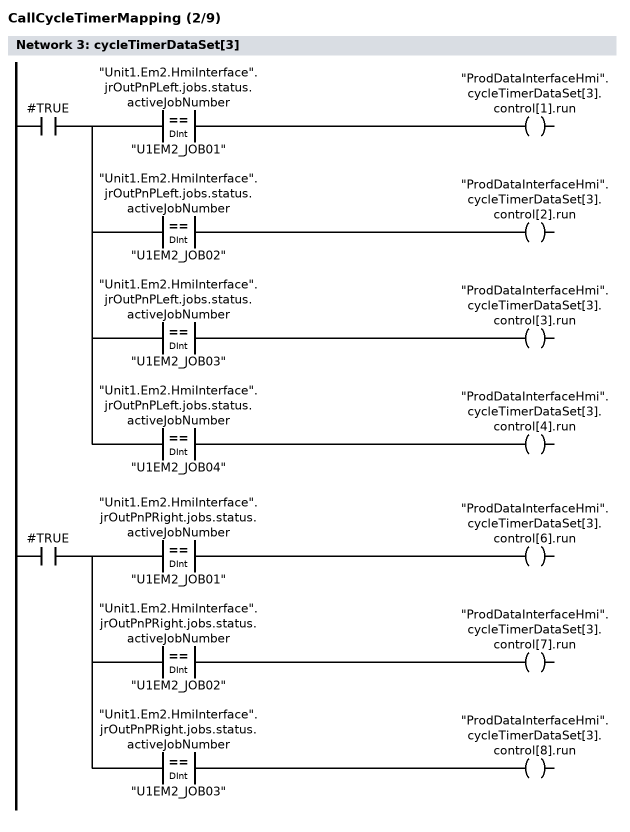
   RUNG wire#powerrail
      Contact( #TRUE )
      wire#w1
      { S7_Templates := "SrcType := DInt" } EQ_Contact(in1 := "Unit1.Em2.HmiInterface".jrOutPnPLeft.jobs.status.activeJobNumber, in2 := "U1EM2_JOB01")
      Coil( "ProdDataInterfaceHmi".cycleTimerDataSet[3].control[1].run )
   END_RUNG
   RUNG wire#w1
      { S7_Templates := "SrcType := DInt" } EQ_Contact(in1 := "Unit1.Em2.HmiInterface".jrOutPnPLeft.jobs.status.activeJobNumber, in2 := "U1EM2_JOB02")
      Coil( "ProdDataInterfaceHmi".cycleTimerDataSet[3].control[2].run )
   END_RUNG
   RUNG wire#w1
      { S7_Templates := "SrcType := DInt" } EQ_Contact(in1 := "Unit1.Em2.HmiInterface".jrOutPnPLeft.jobs.status.activeJobNumber, in2 := "U1EM2_JOB03")
      Coil( "ProdDataInterfaceHmi".cycleTimerDataSet[3].control[3].run )
   END_RUNG
   RUNG wire#w1
      { S7_Templates := "SrcType := DInt" } EQ_Contact(in1 := "Unit1.Em2.HmiInterface".jrOutPnPLeft.jobs.status.activeJobNumber, in2 := "U1EM2_JOB04")
      Coil( "ProdDataInterfaceHmi".cycleTimerDataSet[3].control[4].run )
   END_RUNG
   RUNG wire#powerrail
      Contact( #TRUE )
      wire#w2
      { S7_Templates := "SrcType := DInt" } EQ_Contact(in1 := "Unit1.Em2.HmiInterface".jrOutPnPRight.jobs.status.activeJobNumber, in2 := "U1EM2_JOB01")
      Coil( "ProdDataInterfaceHmi".cycleTimerDataSet[3].control[6].run )
   END_RUNG
   RUNG wire#w2
      { S7_Templates := "SrcType := DInt" } EQ_Contact(in1 := "Unit1.Em2.HmiInterface".jrOutPnPRight.jobs.status.activeJobNumber, in2 := "U1EM2_JOB02")
      Coil( "ProdDataInterfaceHmi".cycleTimerDataSet[3].control[7].run )
   END_RUNG
   RUNG wire#w2
      { S7_Templates := "SrcType := DInt" } EQ_Contact(in1 := "Unit1.Em2.HmiInterface".jrOutPnPRight.jobs.status.activeJobNumber, in2 := "U1EM2_JOB03")
      Coil( "ProdDataInterfaceHmi".cycleTimerDataSet[3].control[8].run )
   END_RUNG
   // the same network as SCL:
   "ProdDataInterfaceHmi".cycleTimerDataSet[3].control[1].run := #TRUE AND ("Unit1.Em2.HmiInterface".jrOutPnPLeft.jobs.status.activeJobNumber = "U1EM2_JOB01");
   "ProdDataInterfaceHmi".cycleTimerDataSet[3].control[2].run := #TRUE AND ("Unit1.Em2.HmiInterface".jrOutPnPLeft.jobs.status.activeJobNumber = "U1EM2_JOB02");
   "ProdDataInterfaceHmi".cycleTimerDataSet[3].control[3].run := #TRUE AND ("Unit1.Em2.HmiInterface".jrOutPnPLeft.jobs.status.activeJobNumber = "U1EM2_JOB03");
   "ProdDataInterfaceHmi".cycleTimerDataSet[3].control[4].run := #TRUE AND ("Unit1.Em2.HmiInterface".jrOutPnPLeft.jobs.status.activeJobNumber = "U1EM2_JOB04");
   "ProdDataInterfaceHmi".cycleTimerDataSet[3].control[6].run := #TRUE AND ("Unit1.Em2.HmiInterface".jrOutPnPRight.jobs.status.activeJobNumber = "U1EM2_JOB01");
   "ProdDataInterfaceHmi".cycleTimerDataSet[3].control[7].run := #TRUE AND ("Unit1.Em2.HmiInterface".jrOutPnPRight.jobs.status.activeJobNumber = "U1EM2_JOB02");
   "ProdDataInterfaceHmi".cycleTimerDataSet[3].control[8].run := #TRUE AND ("Unit1.Em2.HmiInterface".jrOutPnPRight.jobs.status.activeJobNumber = "U1EM2_JOB03");
END_REGION

REGION Network 4: cycleTimerDataSet[4]
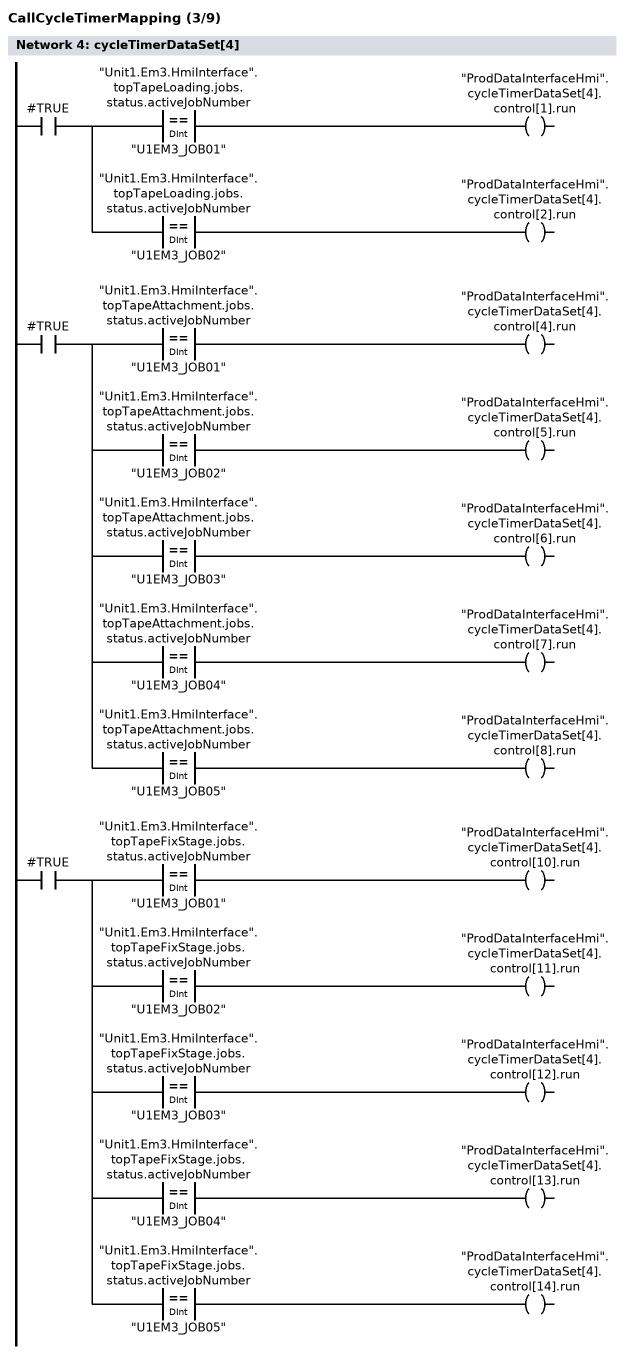
   RUNG wire#powerrail
      Contact( #TRUE )
      wire#w1
      { S7_Templates := "SrcType := DInt" } EQ_Contact(in1 := "Unit1.Em3.HmiInterface".topTapeLoading.jobs.status.activeJobNumber, in2 := "U1EM3_JOB01")
      Coil( "ProdDataInterfaceHmi".cycleTimerDataSet[4].control[1].run )
   END_RUNG
   RUNG wire#w1
      { S7_Templates := "SrcType := DInt" } EQ_Contact(in1 := "Unit1.Em3.HmiInterface".topTapeLoading.jobs.status.activeJobNumber, in2 := "U1EM3_JOB02")
      Coil( "ProdDataInterfaceHmi".cycleTimerDataSet[4].control[2].run )
   END_RUNG
   RUNG wire#powerrail
      Contact( #TRUE )
      wire#w2
      { S7_Templates := "SrcType := DInt" } EQ_Contact(in1 := "Unit1.Em3.HmiInterface".topTapeAttachment.jobs.status.activeJobNumber, in2 := "U1EM3_JOB01")
      Coil( "ProdDataInterfaceHmi".cycleTimerDataSet[4].control[4].run )
   END_RUNG
   RUNG wire#w2
      { S7_Templates := "SrcType := DInt" } EQ_Contact(in1 := "Unit1.Em3.HmiInterface".topTapeAttachment.jobs.status.activeJobNumber, in2 := "U1EM3_JOB02")
      Coil( "ProdDataInterfaceHmi".cycleTimerDataSet[4].control[5].run )
   END_RUNG
   RUNG wire#w2
      { S7_Templates := "SrcType := DInt" } EQ_Contact(in1 := "Unit1.Em3.HmiInterface".topTapeAttachment.jobs.status.activeJobNumber, in2 := "U1EM3_JOB03")
      Coil( "ProdDataInterfaceHmi".cycleTimerDataSet[4].control[6].run )
   END_RUNG
   RUNG wire#w2
      { S7_Templates := "SrcType := DInt" } EQ_Contact(in1 := "Unit1.Em3.HmiInterface".topTapeAttachment.jobs.status.activeJobNumber, in2 := "U1EM3_JOB04")
      Coil( "ProdDataInterfaceHmi".cycleTimerDataSet[4].control[7].run )
   END_RUNG
   RUNG wire#w2
      { S7_Templates := "SrcType := DInt" } EQ_Contact(in1 := "Unit1.Em3.HmiInterface".topTapeAttachment.jobs.status.activeJobNumber, in2 := "U1EM3_JOB05")
      Coil( "ProdDataInterfaceHmi".cycleTimerDataSet[4].control[8].run )
   END_RUNG
   RUNG wire#powerrail
      Contact( #TRUE )
      wire#w3
      { S7_Templates := "SrcType := DInt" } EQ_Contact(in1 := "Unit1.Em3.HmiInterface".topTapeFixStage.jobs.status.activeJobNumber, in2 := "U1EM3_JOB01")
      Coil( "ProdDataInterfaceHmi".cycleTimerDataSet[4].control[10].run )
   END_RUNG
   RUNG wire#w3
      { S7_Templates := "SrcType := DInt" } EQ_Contact(in1 := "Unit1.Em3.HmiInterface".topTapeFixStage.jobs.status.activeJobNumber, in2 := "U1EM3_JOB02")
      Coil( "ProdDataInterfaceHmi".cycleTimerDataSet[4].control[11].run )
   END_RUNG
   RUNG wire#w3
      { S7_Templates := "SrcType := DInt" } EQ_Contact(in1 := "Unit1.Em3.HmiInterface".topTapeFixStage.jobs.status.activeJobNumber, in2 := "U1EM3_JOB03")
      Coil( "ProdDataInterfaceHmi".cycleTimerDataSet[4].control[12].run )
   END_RUNG
   RUNG wire#w3
      { S7_Templates := "SrcType := DInt" } EQ_Contact(in1 := "Unit1.Em3.HmiInterface".topTapeFixStage.jobs.status.activeJobNumber, in2 := "U1EM3_JOB04")
      Coil( "ProdDataInterfaceHmi".cycleTimerDataSet[4].control[13].run )
   END_RUNG
   RUNG wire#w3
      { S7_Templates := "SrcType := DInt" } EQ_Contact(in1 := "Unit1.Em3.HmiInterface".topTapeFixStage.jobs.status.activeJobNumber, in2 := "U1EM3_JOB05")
      Coil( "ProdDataInterfaceHmi".cycleTimerDataSet[4].control[14].run )
   END_RUNG
   // the same network as SCL:
   "ProdDataInterfaceHmi".cycleTimerDataSet[4].control[1].run := #TRUE AND ("Unit1.Em3.HmiInterface".topTapeLoading.jobs.status.activeJobNumber = "U1EM3_JOB01");
   "ProdDataInterfaceHmi".cycleTimerDataSet[4].control[2].run := #TRUE AND ("Unit1.Em3.HmiInterface".topTapeLoading.jobs.status.activeJobNumber = "U1EM3_JOB02");
   "ProdDataInterfaceHmi".cycleTimerDataSet[4].control[4].run := #TRUE AND ("Unit1.Em3.HmiInterface".topTapeAttachment.jobs.status.activeJobNumber = "U1EM3_JOB01");
   "ProdDataInterfaceHmi".cycleTimerDataSet[4].control[5].run := #TRUE AND ("Unit1.Em3.HmiInterface".topTapeAttachment.jobs.status.activeJobNumber = "U1EM3_JOB02");
   "ProdDataInterfaceHmi".cycleTimerDataSet[4].control[6].run := #TRUE AND ("Unit1.Em3.HmiInterface".topTapeAttachment.jobs.status.activeJobNumber = "U1EM3_JOB03");
   "ProdDataInterfaceHmi".cycleTimerDataSet[4].control[7].run := #TRUE AND ("Unit1.Em3.HmiInterface".topTapeAttachment.jobs.status.activeJobNumber = "U1EM3_JOB04");
   "ProdDataInterfaceHmi".cycleTimerDataSet[4].control[8].run := #TRUE AND ("Unit1.Em3.HmiInterface".topTapeAttachment.jobs.status.activeJobNumber = "U1EM3_JOB05");
   "ProdDataInterfaceHmi".cycleTimerDataSet[4].control[10].run := #TRUE AND ("Unit1.Em3.HmiInterface".topTapeFixStage.jobs.status.activeJobNumber = "U1EM3_JOB01");
   "ProdDataInterfaceHmi".cycleTimerDataSet[4].control[11].run := #TRUE AND ("Unit1.Em3.HmiInterface".topTapeFixStage.jobs.status.activeJobNumber = "U1EM3_JOB02");
   "ProdDataInterfaceHmi".cycleTimerDataSet[4].control[12].run := #TRUE AND ("Unit1.Em3.HmiInterface".topTapeFixStage.jobs.status.activeJobNumber = "U1EM3_JOB03");
   "ProdDataInterfaceHmi".cycleTimerDataSet[4].control[13].run := #TRUE AND ("Unit1.Em3.HmiInterface".topTapeFixStage.jobs.status.activeJobNumber = "U1EM3_JOB04");
   "ProdDataInterfaceHmi".cycleTimerDataSet[4].control[14].run := #TRUE AND ("Unit1.Em3.HmiInterface".topTapeFixStage.jobs.status.activeJobNumber = "U1EM3_JOB05");
END_REGION

REGION Network 5: cycleTimerDataSet[5]
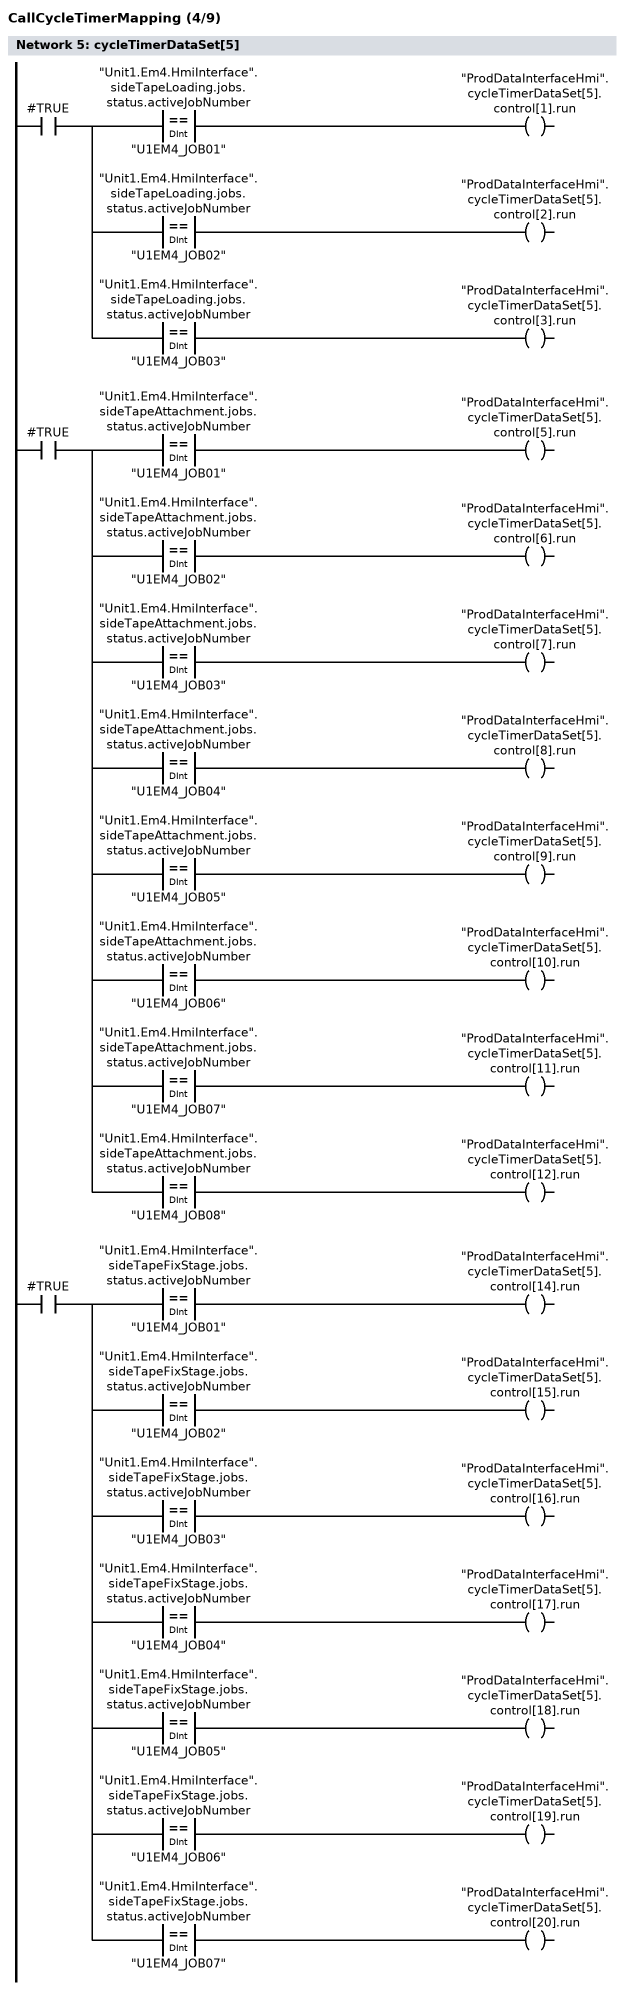
   RUNG wire#powerrail
      Contact( #TRUE )
      wire#w1
      { S7_Templates := "SrcType := DInt" } EQ_Contact(in1 := "Unit1.Em4.HmiInterface".sideTapeLoading.jobs.status.activeJobNumber, in2 := "U1EM4_JOB01")
      Coil( "ProdDataInterfaceHmi".cycleTimerDataSet[5].control[1].run )
   END_RUNG
   RUNG wire#w1
      { S7_Templates := "SrcType := DInt" } EQ_Contact(in1 := "Unit1.Em4.HmiInterface".sideTapeLoading.jobs.status.activeJobNumber, in2 := "U1EM4_JOB02")
      Coil( "ProdDataInterfaceHmi".cycleTimerDataSet[5].control[2].run )
   END_RUNG
   RUNG wire#w1
      { S7_Templates := "SrcType := DInt" } EQ_Contact(in1 := "Unit1.Em4.HmiInterface".sideTapeLoading.jobs.status.activeJobNumber, in2 := "U1EM4_JOB03")
      Coil( "ProdDataInterfaceHmi".cycleTimerDataSet[5].control[3].run )
   END_RUNG
   RUNG wire#powerrail
      Contact( #TRUE )
      wire#w2
      { S7_Templates := "SrcType := DInt" } EQ_Contact(in1 := "Unit1.Em4.HmiInterface".sideTapeAttachment.jobs.status.activeJobNumber, in2 := "U1EM4_JOB01")
      Coil( "ProdDataInterfaceHmi".cycleTimerDataSet[5].control[5].run )
   END_RUNG
   RUNG wire#w2
      { S7_Templates := "SrcType := DInt" } EQ_Contact(in1 := "Unit1.Em4.HmiInterface".sideTapeAttachment.jobs.status.activeJobNumber, in2 := "U1EM4_JOB02")
      Coil( "ProdDataInterfaceHmi".cycleTimerDataSet[5].control[6].run )
   END_RUNG
   RUNG wire#w2
      { S7_Templates := "SrcType := DInt" } EQ_Contact(in1 := "Unit1.Em4.HmiInterface".sideTapeAttachment.jobs.status.activeJobNumber, in2 := "U1EM4_JOB03")
      Coil( "ProdDataInterfaceHmi".cycleTimerDataSet[5].control[7].run )
   END_RUNG
   RUNG wire#w2
      { S7_Templates := "SrcType := DInt" } EQ_Contact(in1 := "Unit1.Em4.HmiInterface".sideTapeAttachment.jobs.status.activeJobNumber, in2 := "U1EM4_JOB04")
      Coil( "ProdDataInterfaceHmi".cycleTimerDataSet[5].control[8].run )
   END_RUNG
   RUNG wire#w2
      { S7_Templates := "SrcType := DInt" } EQ_Contact(in1 := "Unit1.Em4.HmiInterface".sideTapeAttachment.jobs.status.activeJobNumber, in2 := "U1EM4_JOB05")
      Coil( "ProdDataInterfaceHmi".cycleTimerDataSet[5].control[9].run )
   END_RUNG
   RUNG wire#w2
      { S7_Templates := "SrcType := DInt" } EQ_Contact(in1 := "Unit1.Em4.HmiInterface".sideTapeAttachment.jobs.status.activeJobNumber, in2 := "U1EM4_JOB06")
      Coil( "ProdDataInterfaceHmi".cycleTimerDataSet[5].control[10].run )
   END_RUNG
   RUNG wire#w2
      { S7_Templates := "SrcType := DInt" } EQ_Contact(in1 := "Unit1.Em4.HmiInterface".sideTapeAttachment.jobs.status.activeJobNumber, in2 := "U1EM4_JOB07")
      Coil( "ProdDataInterfaceHmi".cycleTimerDataSet[5].control[11].run )
   END_RUNG
   RUNG wire#w2
      { S7_Templates := "SrcType := DInt" } EQ_Contact(in1 := "Unit1.Em4.HmiInterface".sideTapeAttachment.jobs.status.activeJobNumber, in2 := "U1EM4_JOB08")
      Coil( "ProdDataInterfaceHmi".cycleTimerDataSet[5].control[12].run )
   END_RUNG
   RUNG wire#powerrail
      Contact( #TRUE )
      wire#w3
      { S7_Templates := "SrcType := DInt" } EQ_Contact(in1 := "Unit1.Em4.HmiInterface".sideTapeFixStage.jobs.status.activeJobNumber, in2 := "U1EM4_JOB01")
      Coil( "ProdDataInterfaceHmi".cycleTimerDataSet[5].control[14].run )
   END_RUNG
   RUNG wire#w3
      { S7_Templates := "SrcType := DInt" } EQ_Contact(in1 := "Unit1.Em4.HmiInterface".sideTapeFixStage.jobs.status.activeJobNumber, in2 := "U1EM4_JOB02")
      Coil( "ProdDataInterfaceHmi".cycleTimerDataSet[5].control[15].run )
   END_RUNG
   RUNG wire#w3
      { S7_Templates := "SrcType := DInt" } EQ_Contact(in1 := "Unit1.Em4.HmiInterface".sideTapeFixStage.jobs.status.activeJobNumber, in2 := "U1EM4_JOB03")
      Coil( "ProdDataInterfaceHmi".cycleTimerDataSet[5].control[16].run )
   END_RUNG
   RUNG wire#w3
      { S7_Templates := "SrcType := DInt" } EQ_Contact(in1 := "Unit1.Em4.HmiInterface".sideTapeFixStage.jobs.status.activeJobNumber, in2 := "U1EM4_JOB04")
      Coil( "ProdDataInterfaceHmi".cycleTimerDataSet[5].control[17].run )
   END_RUNG
   RUNG wire#w3
      { S7_Templates := "SrcType := DInt" } EQ_Contact(in1 := "Unit1.Em4.HmiInterface".sideTapeFixStage.jobs.status.activeJobNumber, in2 := "U1EM4_JOB05")
      Coil( "ProdDataInterfaceHmi".cycleTimerDataSet[5].control[18].run )
   END_RUNG
   RUNG wire#w3
      { S7_Templates := "SrcType := DInt" } EQ_Contact(in1 := "Unit1.Em4.HmiInterface".sideTapeFixStage.jobs.status.activeJobNumber, in2 := "U1EM4_JOB06")
      Coil( "ProdDataInterfaceHmi".cycleTimerDataSet[5].control[19].run )
   END_RUNG
   RUNG wire#w3
      { S7_Templates := "SrcType := DInt" } EQ_Contact(in1 := "Unit1.Em4.HmiInterface".sideTapeFixStage.jobs.status.activeJobNumber, in2 := "U1EM4_JOB07")
      Coil( "ProdDataInterfaceHmi".cycleTimerDataSet[5].control[20].run )
   END_RUNG
   // the same network as SCL:
   "ProdDataInterfaceHmi".cycleTimerDataSet[5].control[1].run := #TRUE AND ("Unit1.Em4.HmiInterface".sideTapeLoading.jobs.status.activeJobNumber = "U1EM4_JOB01");
   "ProdDataInterfaceHmi".cycleTimerDataSet[5].control[2].run := #TRUE AND ("Unit1.Em4.HmiInterface".sideTapeLoading.jobs.status.activeJobNumber = "U1EM4_JOB02");
   "ProdDataInterfaceHmi".cycleTimerDataSet[5].control[3].run := #TRUE AND ("Unit1.Em4.HmiInterface".sideTapeLoading.jobs.status.activeJobNumber = "U1EM4_JOB03");
   "ProdDataInterfaceHmi".cycleTimerDataSet[5].control[5].run := #TRUE AND ("Unit1.Em4.HmiInterface".sideTapeAttachment.jobs.status.activeJobNumber = "U1EM4_JOB01");
   "ProdDataInterfaceHmi".cycleTimerDataSet[5].control[6].run := #TRUE AND ("Unit1.Em4.HmiInterface".sideTapeAttachment.jobs.status.activeJobNumber = "U1EM4_JOB02");
   "ProdDataInterfaceHmi".cycleTimerDataSet[5].control[7].run := #TRUE AND ("Unit1.Em4.HmiInterface".sideTapeAttachment.jobs.status.activeJobNumber = "U1EM4_JOB03");
   "ProdDataInterfaceHmi".cycleTimerDataSet[5].control[8].run := #TRUE AND ("Unit1.Em4.HmiInterface".sideTapeAttachment.jobs.status.activeJobNumber = "U1EM4_JOB04");
   "ProdDataInterfaceHmi".cycleTimerDataSet[5].control[9].run := #TRUE AND ("Unit1.Em4.HmiInterface".sideTapeAttachment.jobs.status.activeJobNumber = "U1EM4_JOB05");
   "ProdDataInterfaceHmi".cycleTimerDataSet[5].control[10].run := #TRUE AND ("Unit1.Em4.HmiInterface".sideTapeAttachment.jobs.status.activeJobNumber = "U1EM4_JOB06");
   "ProdDataInterfaceHmi".cycleTimerDataSet[5].control[11].run := #TRUE AND ("Unit1.Em4.HmiInterface".sideTapeAttachment.jobs.status.activeJobNumber = "U1EM4_JOB07");
   "ProdDataInterfaceHmi".cycleTimerDataSet[5].control[12].run := #TRUE AND ("Unit1.Em4.HmiInterface".sideTapeAttachment.jobs.status.activeJobNumber = "U1EM4_JOB08");
   "ProdDataInterfaceHmi".cycleTimerDataSet[5].control[14].run := #TRUE AND ("Unit1.Em4.HmiInterface".sideTapeFixStage.jobs.status.activeJobNumber = "U1EM4_JOB01");
   "ProdDataInterfaceHmi".cycleTimerDataSet[5].control[15].run := #TRUE AND ("Unit1.Em4.HmiInterface".sideTapeFixStage.jobs.status.activeJobNumber = "U1EM4_JOB02");
   "ProdDataInterfaceHmi".cycleTimerDataSet[5].control[16].run := #TRUE AND ("Unit1.Em4.HmiInterface".sideTapeFixStage.jobs.status.activeJobNumber = "U1EM4_JOB03");
   "ProdDataInterfaceHmi".cycleTimerDataSet[5].control[17].run := #TRUE AND ("Unit1.Em4.HmiInterface".sideTapeFixStage.jobs.status.activeJobNumber = "U1EM4_JOB04");
   "ProdDataInterfaceHmi".cycleTimerDataSet[5].control[18].run := #TRUE AND ("Unit1.Em4.HmiInterface".sideTapeFixStage.jobs.status.activeJobNumber = "U1EM4_JOB05");
   "ProdDataInterfaceHmi".cycleTimerDataSet[5].control[19].run := #TRUE AND ("Unit1.Em4.HmiInterface".sideTapeFixStage.jobs.status.activeJobNumber = "U1EM4_JOB06");
   "ProdDataInterfaceHmi".cycleTimerDataSet[5].control[20].run := #TRUE AND ("Unit1.Em4.HmiInterface".sideTapeFixStage.jobs.status.activeJobNumber = "U1EM4_JOB07");
END_REGION

